LIN {X -0.230,Y -500.560,Z 1588.535,A 0.000,B 0.000,C 90.000,E1 96.372} C_DIS
LIN {X 0.139,Y -499.439,Z 1588.534,A 0.000,B 0.000,C 90.000,E1 96.087} C_DIS
LIN {X -0.151,Y -494.579,Z 1588.530,A 0.000,B 0.000,C 90.000,E1 95.391} C_DIS
LIN {X 0.194,Y -481.570,Z 1588.519,A 0.000,B 0.000,C 90.000,E1 93.383} C_DIS
LIN {X 0.131,Y -471.581,Z 1588.511,A 0.000,B 0.000,C 90.000,E1 91.892} C_DIS
LIN {X 0.103,Y -462.930,Z 1588.504,A 0.000,B 0.000,C 90.000,E1 90.630} C_DIS
LIN {X -0.051,Y -453.933,Z 1588.496,A 0.000,B 0.000,C 90.000,E1 89.370} C_DIS
LIN {X 0.124,Y -444.506,Z 1588.489,A 0.000,B 0.000,C 90.000,E1 88.051} C_DIS
LIN {X -0.111,Y -432.606,Z 1588.480,A 0.000,B 0.000,C 90.000,E1 86.502} C_DIS
LIN {X 0.018,Y -418.492,Z 1588.470,A 0.000,B 0.000,C 90.000,E1 84.609} C_DIS
LIN {X 0.166,Y -399.403,Z 1588.455,A 0.000,B 0.000,C 90.000,E1 81.837} C_DIS
LIN {X -0.155,Y -383.351,Z 1588.441,A 0.000,B 0.000,C 90.000,E1 79.342} C_DIS
LIN {X 0.055,Y -364.882,Z 1588.423,A 0.000,B 0.000,C 90.000,E1 76.117} C_DIS
LIN {X 0.022,Y -351.994,Z 1588.410,A 0.000,B 0.000,C 90.000,E1 73.740} C_DIS
LIN {X -0.111,Y -339.351,Z 1588.396,A 0.000,B 0.000,C 90.000,E1 71.329} C_DIS
LIN {X -0.034,Y -325.790,Z 1588.381,A 0.000,B 0.000,C 90.000,E1 68.518} C_DIS
LIN {X -0.019,Y -314.232,Z 1588.366,A 0.000,B 0.000,C 90.000,E1 65.973} C_DIS
LIN {X -0.119,Y -300.650,Z 1588.348,A 0.000,B 0.000,C 90.000,E1 62.743} C_DIS
LIN {X 0.080,Y -292.540,Z 1588.337,A 0.000,B 0.000,C 90.000,E1 60.717} C_DIS
LIN {X -0.130,Y -284.116,Z 1588.326,A 0.000,B 0.000,C 90.000,E1 58.742} C_DIS
LIN {X 0.132,Y -273.947,Z 1588.313,A 0.000,B 0.000,C 90.000,E1 56.294} C_DIS
LIN {X -0.133,Y -263.749,Z 1588.299,A 0.000,B 0.000,C 90.000,E1 53.909} C_DIS
LIN {X -0.023,Y -251.335,Z 1588.281,A 0.000,B 0.000,C 90.000,E1 50.678} C_DIS
LIN {X -0.018,Y -239.866,Z 1588.263,A 0.000,B 0.000,C 90.000,E1 47.391} C_DIS
LIN {X -0.003,Y -229.485,Z 1588.245,A 0.000,B 0.000,C 90.000,E1 44.028} C_DIS
LIN {X -0.004,Y -221.059,Z 1588.228,A 0.000,B 0.000,C 90.000,E1 40.987} C_DIS
LIN {X 0.009,Y -213.332,Z 1588.211,A 0.000,B 0.000,C 90.000,E1 37.890} C_DIS
LIN {X 0.035,Y -206.409,Z 1588.193,A 0.000,B 0.000,C 90.000,E1 34.739} C_DIS
LIN {X 0.050,Y -200.208,Z 1588.175,A 0.000,B 0.000,C 90.000,E1 31.544} C_DIS
LIN {X 0.055,Y -194.851,Z 1588.157,A 0.000,B 0.000,C 90.000,E1 28.309} C_DIS
LIN {X 0.086,Y -190.223,Z 1588.139,A 0.000,B 0.000,C 90.000,E1 25.027} C_DIS
LIN {X -0.003,Y -185.282,Z 1588.116,A 0.000,B 0.000,C 90.000,E1 20.918} C_DIS
LIN {X 0.013,Y -181.201,Z 1588.093,A 0.000,B 0.000,C 90.000,E1 16.732} C_DIS
LIN {X -0.054,Y -177.876,Z 1588.070,A 0.000,B 0.000,C 90.000,E1 12.535} C_DIS
LIN {X 0.018,Y -175.021,Z 1588.041,A 0.000,B 0.000,C 90.000,E1 7.409} C_DIS
LIN {X -0.025,Y -172.799,Z 1588.008,A 0.000,B 0.000,C 90.000,E1 1.432} C_DIS
LIN {X 0.049,Y -173.988,Z 1587.935,A 0.000,B 0.000,C 90.000,E1 348.342} C_DIS
LIN {X 0.090,Y -176.815,Z 1587.907,A 0.000,B 0.000,C 90.000,E1 343.196} C_DIS
LIN {X 0.073,Y -180.404,Z 1587.883,A 0.000,B 0.000,C 90.000,E1 338.954} C_DIS
LIN {X -0.083,Y -185.209,Z 1587.860,A 0.000,B 0.000,C 90.000,E1 334.793} C_DIS
LIN {X -0.009,Y -189.881,Z 1587.841,A 0.000,B 0.000,C 90.000,E1 331.435} C_DIS
LIN {X 0.040,Y -195.211,Z 1587.823,A 0.000,B 0.000,C 90.000,E1 328.122} C_DIS
LIN {X -0.072,Y -201.335,Z 1587.805,A 0.000,B 0.000,C 90.000,E1 324.895} C_DIS
LIN {X -0.008,Y -208.216,Z 1587.787,A 0.000,B 0.000,C 90.000,E1 321.662} C_DIS
LIN {X 0.040,Y -216.014,Z 1587.769,A 0.000,B 0.000,C 90.000,E1 318.485} C_DIS
LIN {X 0.023,Y -225.787,Z 1587.750,A 0.000,B 0.000,C 90.000,E1 315.000} C_DIS
LIN {X -0.103,Y -234.279,Z 1587.735,A 0.000,B 0.000,C 90.000,E1 312.366} C_DIS
LIN {X 0.012,Y -242.255,Z 1587.723,A 0.000,B 0.000,C 90.000,E1 310.092} C_DIS
LIN {X -0.029,Y -248.230,Z 1587.715,A 0.000,B 0.000,C 90.000,E1 308.624} C_DIS
LIN {X 0.005,Y -254.959,Z 1587.706,A 0.000,B 0.000,C 90.000,E1 307.156} C_DIS
LIN {X 0.013,Y -264.367,Z 1587.696,A 0.000,B 0.000,C 90.000,E1 305.358} C_DIS
LIN {X 0.011,Y -276.846,Z 1587.685,A 0.000,B 0.000,C 90.000,E1 303.245} C_DIS
LIN {X -0.005,Y -293.095,Z 1587.671,A 0.000,B 0.000,C 90.000,E1 300.846} C_DIS
LIN {X 0.122,Y -308.007,Z 1587.660,A 0.000,B 0.000,C 90.000,E1 298.821} C_DIS
LIN {X 0.062,Y -320.406,Z 1587.651,A 0.000,B 0.000,C 90.000,E1 297.206} C_DIS
LIN {X 0.191,Y -332.863,Z 1587.642,A 0.000,B 0.000,C 90.000,E1 295.591} C_DIS
LIN {X -0.075,Y -344.944,Z 1587.634,A 0.000,B 0.000,C 90.000,E1 294.079} C_DIS
LIN {X -0.087,Y -362.411,Z 1587.622,A 0.000,B 0.000,C 90.000,E1 291.950} C_DIS
LIN {X 0.161,Y -374.913,Z 1587.614,A 0.000,B 0.000,C 90.000,E1 290.429} C_DIS
LIN {X 0.128,Y -384.438,Z 1587.607,A 0.000,B 0.000,C 90.000,E1 289.268} C_DIS
LIN {X 0.049,Y -391.088,Z 1587.602,A 0.000,B 0.000,C 90.000,E1 288.417} C_DIS
LIN {X -0.087,Y -397.218,Z 1587.598,A 0.000,B 0.000,C 90.000,E1 287.583} C_DIS
LIN {X 0.148,Y -400.979,Z 1587.594,A 0.000,B 0.000,C 90.000,E1 286.985} C_DIS
LIN {X 0.104,Y -405.869,Z 1587.590,A 0.000,B 0.000,C 90.000,E1 286.150} C_DIS
LIN {X 0.006,Y -408.632,Z 1587.587,A 0.000,B 0.000,C 90.000,E1 285.607} C_DIS
LIN {X -0.077,Y -411.045,Z 1587.584,A 0.000,B 0.000,C 90.000,E1 285.064} C_DIS
LIN {X 0.146,Y -413.036,Z 1587.581,A 0.000,B 0.000,C 90.000,E1 284.481} C_DIS
LIN {X 0.080,Y -414.633,Z 1587.578,A 0.000,B 0.000,C 90.000,E1 283.939} C_DIS
LIN {X -0.077,Y -415.820,Z 1587.574,A 0.000,B 0.000,C 90.000,E1 283.411} C_DIS
LIN {X 0.182,Y -416.599,Z 1587.571,A 0.000,B 0.000,C 90.000,E1 282.827} C_DIS
LIN {X 0.044,Y -416.869,Z 1587.568,A 0.000,B 0.000,C 90.000,E1 282.299} C_DIS
LIN {X -0.090,Y -416.664,Z 1587.565,A 0.000,B 0.000,C 90.000,E1 281.771} C_DIS
LIN {X 0.185,Y -415.926,Z 1587.562,A 0.000,B 0.000,C 90.000,E1 281.186} C_DIS
LIN {X 0.049,Y -414.668,Z 1587.559,A 0.000,B 0.000,C 90.000,E1 280.658} C_DIS
LIN {X -0.165,Y -412.786,Z 1587.556,A 0.000,B 0.000,C 90.000,E1 280.141} C_DIS
LIN {X 0.094,Y -410.280,Z 1587.553,A 0.000,B 0.000,C 90.000,E1 279.557} C_DIS
LIN {X -0.073,Y -407.020,Z 1587.550,A 0.000,B 0.000,C 90.000,E1 279.029} C_DIS
LIN {X -0.026,Y -405.197,Z 1587.549,A 0.000,B 0.000,C 90.000,E1 278.746} C_DIS
LIN {X 0.177,Y -400.827,Z 1587.546,A 0.000,B 0.000,C 90.000,E1 278.163} C_DIS
LIN {X -0.097,Y -395.813,Z 1587.542,A 0.000,B 0.000,C 90.000,E1 277.644} C_DIS
LIN {X 0.138,Y -390.224,Z 1587.539,A 0.000,B 0.000,C 90.000,E1 277.068} C_DIS
LIN {X -0.161,Y -384.400,Z 1587.537,A 0.000,B 0.000,C 90.000,E1 276.606} C_DIS
LIN {X 0.160,Y -378.276,Z 1587.534,A 0.000,B 0.000,C 90.000,E1 276.087} C_DIS
LIN {X 0.005,Y -371.989,Z 1587.532,A 0.000,B 0.000,C 90.000,E1 275.682} C_DIS
LIN {X 0.032,Y -362.421,Z 1587.528,A 0.000,B 0.000,C 90.000,E1 275.106} C_DIS
LIN {X 0.140,Y -352.870,Z 1587.526,A 0.000,B 0.000,C 90.000,E1 274.588} C_DIS
LIN {X 0.138,Y -343.087,Z 1587.523,A 0.000,B 0.000,C 90.000,E1 274.131} C_DIS
LIN {X 0.113,Y -333.414,Z 1587.521,A 0.000,B 0.000,C 90.000,E1 273.726} C_DIS
LIN {X -0.095,Y -320.424,Z 1587.518,A 0.000,B 0.000,C 90.000,E1 273.269} C_DIS
LIN {X -0.022,Y -310.456,Z 1587.516,A 0.000,B 0.000,C 90.000,E1 272.922} C_DIS
LIN {X -0.024,Y -299.914,Z 1587.515,A 0.000,B 0.000,C 90.000,E1 272.636} C_DIS
LIN {X 0.033,Y -292.289,Z 1587.514,A 0.000,B 0.000,C 90.000,E1 272.465} C_DIS
LIN {X -0.085,Y -279.300,Z 1587.513,A 0.000,B 0.000,C 90.000,E1 272.293} C_DIS
LIN {X -0.016,Y -260.975,Z 1587.511,A 0.000,B 0.000,C 90.000,E1 272.064} C_DIS
LIN {X -0.040,Y -244.011,Z 1587.511,A 0.000,B 0.000,C 90.000,E1 271.949} C_DIS
LIN {X 0.107,Y -235.308,Z 1587.511,A 0.000,B 0.000,C 90.000,E1 271.892} C_DIS
LIN {X 0.048,Y -181.277,Z 1587.511,A 0.000,B 0.000,C 90.000,E1 271.892} C_DIS
LIN {X 0.057,Y -181.579,Z 1587.501,A 0.000,B 0.000,C 90.000,E1 270.172} C_DIS
LIN {X 0.045,Y -180.887,Z 1587.473,A 0.000,B 0.000,C 90.000,E1 265.122} C_DIS
LIN {X -0.072,Y -179.010,Z 1587.445,A 0.000,B 0.000,C 90.000,E1 260.095} C_DIS
LIN {X 0.023,Y -178.625,Z 1587.440,A 0.000,B 0.000,C 90.000,E1 259.218} C_DIS
LIN {X -0.079,Y -175.676,Z 1587.412,A 0.000,B 0.000,C 90.000,E1 254.157} C_DIS
LIN {X -0.067,Y -172.393,Z 1587.388,A 0.000,B 0.000,C 90.000,E1 249.880} C_DIS
LIN {X -0.050,Y -171.199,Z 1587.379,A 0.000,B 0.000,C 90.000,E1 248.156} C_DIS
LIN {X 0.001,Y -167.488,Z 1587.355,A 0.000,B 0.000,C 90.000,E1 243.819} C_DIS
LIN {X 0.009,Y -166.884,Z 1587.350,A 0.000,B 0.000,C 90.000,E1 242.948} C_DIS
LIN {X 0.000,Y -162.189,Z 1587.321,A 0.000,B 0.000,C 90.000,E1 237.709} C_DIS
LIN {X -0.033,Y -160.758,Z 1587.311,A 0.000,B 0.000,C 90.000,E1 235.960} C_DIS
LIN {X 0.036,Y -157.555,Z 1587.291,A 0.000,B 0.000,C 90.000,E1 232.396} C_DIS
LIN {X -0.027,Y -155.584,Z 1587.276,A 0.000,B 0.000,C 90.000,E1 229.747} C_DIS
LIN {X 0.025,Y -151.869,Z 1587.251,A 0.000,B 0.000,C 90.000,E1 225.243} C_DIS
LIN {X 0.039,Y -150.093,Z 1587.236,A 0.000,B 0.000,C 90.000,E1 222.528} C_DIS
LIN {X -0.044,Y -146.893,Z 1587.211,A 0.000,B 0.000,C 90.000,E1 218.016} C_DIS
LIN {X 0.061,Y -145.480,Z 1587.196,A 0.000,B 0.000,C 90.000,E1 215.231} C_DIS
LIN {X -0.023,Y -142.889,Z 1587.170,A 0.000,B 0.000,C 90.000,E1 210.669} C_DIS
LIN {X 0.034,Y -141.509,Z 1587.150,A 0.000,B 0.000,C 90.000,E1 206.950} C_DIS
LIN {X -0.049,Y -139.391,Z 1587.114,A 0.000,B 0.000,C 90.000,E1 200.482} C_DIS
LIN {X 0.003,Y -139.100,Z 1587.103,A 0.000,B 0.000,C 90.000,E1 198.598} C_DIS
LIN {X -0.006,Y -138.353,Z 1587.057,A 0.000,B 0.000,C 90.000,E1 190.197} C_DIS
LIN {X -0.012,Y -139.515,Z 1587.005,A 0.000,B 0.000,C 90.000,E1 180.859} C_DIS
LIN {X -0.072,Y -141.166,Z 1586.974,A 0.000,B 0.000,C 90.000,E1 175.298} C_DIS
LIN {X 0.040,Y -142.545,Z 1586.958,A 0.000,B 0.000,C 90.000,E1 172.470} C_DIS
LIN {X -0.035,Y -144.819,Z 1586.933,A 0.000,B 0.000,C 90.000,E1 167.881} C_DIS
LIN {X -0.048,Y -147.440,Z 1586.912,A 0.000,B 0.000,C 90.000,E1 164.212} C_DIS
LIN {X -0.019,Y -150.020,Z 1586.892,A 0.000,B 0.000,C 90.000,E1 160.550} C_DIS
LIN {X -0.013,Y -153.355,Z 1586.872,A 0.000,B 0.000,C 90.000,E1 156.922} C_DIS
LIN {X 0.036,Y -155.889,Z 1586.857,A 0.000,B 0.000,C 90.000,E1 154.204} C_DIS
LIN {X -0.066,Y -159.746,Z 1586.837,A 0.000,B 0.000,C 90.000,E1 150.667} C_DIS
LIN {X 0.000,Y -161.987,Z 1586.827,A 0.000,B 0.000,C 90.000,E1 148.869} C_DIS
LIN {X 0.020,Y -166.179,Z 1586.807,A 0.000,B 0.000,C 90.000,E1 145.341} C_DIS
LIN {X 0.013,Y -171.193,Z 1586.788,A 0.000,B 0.000,C 90.000,E1 141.859} C_DIS
LIN {X 0.043,Y -176.076,Z 1586.769,A 0.000,B 0.000,C 90.000,E1 138.405} C_DIS
LIN {X -0.094,Y -180.335,Z 1586.755,A 0.000,B 0.000,C 90.000,E1 135.891} C_DIS
LIN {X 0.014,Y -185.744,Z 1586.736,A 0.000,B 0.000,C 90.000,E1 132.486} C_DIS
LIN {X -0.073,Y -190.355,Z 1586.722,A 0.000,B 0.000,C 90.000,E1 130.011} C_DIS
LIN {X -0.026,Y -197.681,Z 1586.699,A 0.000,B 0.000,C 90.000,E1 125.884} C_DIS
LIN {X 0.015,Y -200.933,Z 1586.690,A 0.000,B 0.000,C 90.000,E1 124.246} C_DIS
LIN {X 0.074,Y -204.518,Z 1586.679,A 0.000,B 0.000,C 90.000,E1 122.212} C_DIS
LIN {X 0.056,Y -322.284,Z 1586.679,A 0.000,B 0.000,C 90.000,E1 122.212} C_DIS
LIN {X -0.123,Y -323.983,Z 1586.679,A 0.000,B 0.000,C 90.000,E1 122.212} C_DIS
LIN {X 0.034,Y -327.982,Z 1586.678,A 0.000,B 0.000,C 90.000,E1 122.005} C_DIS
LIN {X 0.193,Y -330.311,Z 1586.677,A 0.000,B 0.000,C 90.000,E1 121.799} C_DIS
LIN {X -0.018,Y -334.169,Z 1586.674,A 0.000,B 0.000,C 90.000,E1 121.386} C_DIS
LIN {X 0.129,Y -336.011,Z 1586.673,A 0.000,B 0.000,C 90.000,E1 121.052} C_DIS
LIN {X -0.047,Y -338.678,Z 1586.669,A 0.000,B 0.000,C 90.000,E1 120.463} C_DIS
LIN {X -0.038,Y -350.483,Z 1586.654,A 0.000,B 0.000,C 90.000,E1 117.692} C_DIS
LIN {X 0.139,Y -363.724,Z 1586.639,A 0.000,B 0.000,C 90.000,E1 114.951} C_DIS
LIN {X -0.094,Y -378.522,Z 1586.624,A 0.000,B 0.000,C 90.000,E1 112.333} C_DIS
LIN {X 0.143,Y -393.083,Z 1586.611,A 0.000,B 0.000,C 90.000,E1 109.993} C_DIS
LIN {X -0.023,Y -409.073,Z 1586.599,A 0.000,B 0.000,C 90.000,E1 107.764} C_DIS
LIN {X 0.089,Y -426.603,Z 1586.586,A 0.000,B 0.000,C 90.000,E1 105.552} C_DIS
LIN {X 0.128,Y -445.761,Z 1586.575,A 0.000,B 0.000,C 90.000,E1 103.411} C_DIS
LIN {X 0.086,Y -465.835,Z 1586.563,A 0.000,B 0.000,C 90.000,E1 101.422} C_DIS
LIN {X 0.034,Y -489.042,Z 1586.552,A 0.000,B 0.000,C 90.000,E1 99.378} C_DIS
LIN {X -0.187,Y -494.277,Z 1586.550,A 0.000,B 0.000,C 90.000,E1 98.973} C_DIS
LIN {X -0.072,Y -496.442,Z 1586.549,A 0.000,B 0.000,C 90.000,E1 98.746} C_DIS
LIN {X -0.113,Y -498.267,Z 1586.547,A 0.000,B 0.000,C 90.000,E1 98.511} C_DIS
LIN {X -0.155,Y -499.640,Z 1586.546,A 0.000,B 0.000,C 90.000,E1 98.276} C_DIS
LIN {X 0.118,Y -501.397,Z 1586.543,A 0.000,B 0.000,C 90.000,E1 97.757} C_DIS
LIN {X -0.098,Y -502.041,Z 1586.541,A 0.000,B 0.000,C 90.000,E1 97.296} C_DIS
LIN {X 0.195,Y -501.682,Z 1586.538,A 0.000,B 0.000,C 90.000,E1 96.777} C_DIS
LIN {X -0.006,Y -500.267,Z 1586.535,A 0.000,B 0.000,C 90.000,E1 96.315} C_DIS
LIN {X -0.133,Y -499.089,Z 1586.534,A 0.000,B 0.000,C 90.000,E1 96.087} C_DIS
LIN {X -0.126,Y -486.046,Z 1586.523,A 0.000,B 0.000,C 90.000,E1 94.131} C_DIS
LIN {X -0.083,Y -476.250,Z 1586.515,A 0.000,B 0.000,C 90.000,E1 92.636} C_DIS
LIN {X 0.231,Y -466.095,Z 1586.506,A 0.000,B 0.000,C 90.000,E1 91.088} C_DIS
LIN {X -0.105,Y -455.371,Z 1586.498,A 0.000,B 0.000,C 90.000,E1 89.599} C_DIS
LIN {X 0.083,Y -446.043,Z 1586.490,A 0.000,B 0.000,C 90.000,E1 88.282} C_DIS
LIN {X 0.135,Y -436.232,Z 1586.483,A 0.000,B 0.000,C 90.000,E1 86.963} C_DIS
LIN {X -0.059,Y -422.140,Z 1586.473,A 0.000,B 0.000,C 90.000,E1 85.122} C_DIS
LIN {X -0.198,Y -400.891,Z 1586.456,A 0.000,B 0.000,C 90.000,E1 82.129} C_DIS
LIN {X -0.047,Y -383.024,Z 1586.440,A 0.000,B 0.000,C 90.000,E1 79.285} C_DIS
LIN {X 0.144,Y -364.572,Z 1586.423,A 0.000,B 0.000,C 90.000,E1 76.061} C_DIS
LIN {X 0.095,Y -351.683,Z 1586.409,A 0.000,B 0.000,C 90.000,E1 73.685} C_DIS
LIN {X -0.051,Y -339.047,Z 1586.396,A 0.000,B 0.000,C 90.000,E1 71.275} C_DIS
LIN {X 0.009,Y -325.528,Z 1586.380,A 0.000,B 0.000,C 90.000,E1 68.465} C_DIS
LIN {X 0.011,Y -313.943,Z 1586.366,A 0.000,B 0.000,C 90.000,E1 65.921} C_DIS
LIN {X 0.009,Y -301.647,Z 1586.350,A 0.000,B 0.000,C 90.000,E1 62.999} C_DIS
LIN {X 0.081,Y -293.519,Z 1586.339,A 0.000,B 0.000,C 90.000,E1 61.001} C_DIS
LIN {X 0.030,Y -285.091,Z 1586.328,A 0.000,B 0.000,C 90.000,E1 58.997} C_DIS
LIN {X -0.021,Y -276.443,Z 1586.316,A 0.000,B 0.000,C 90.000,E1 56.962} C_DIS
LIN {X -0.004,Y -266.311,Z 1586.303,A 0.000,B 0.000,C 90.000,E1 54.529} C_DIS
LIN {X 0.022,Y -253.756,Z 1586.285,A 0.000,B 0.000,C 90.000,E1 51.331} C_DIS
LIN {X -0.066,Y -242.103,Z 1586.267,A 0.000,B 0.000,C 90.000,E1 48.081} C_DIS
LIN {X 0.015,Y -231.529,Z 1586.248,A 0.000,B 0.000,C 90.000,E1 44.717} C_DIS
LIN {X 0.052,Y -222.941,Z 1586.232,A 0.000,B 0.000,C 90.000,E1 41.676} C_DIS
LIN {X -0.057,Y -215.065,Z 1586.214,A 0.000,B 0.000,C 90.000,E1 38.624} C_DIS
LIN {X 0.019,Y -207.965,Z 1586.197,A 0.000,B 0.000,C 90.000,E1 35.471} C_DIS
LIN {X 0.020,Y -201.641,Z 1586.179,A 0.000,B 0.000,C 90.000,E1 32.291} C_DIS
LIN {X -0.013,Y -196.095,Z 1586.161,A 0.000,B 0.000,C 90.000,E1 29.077} C_DIS
LIN {X 0.049,Y -191.343,Z 1586.143,A 0.000,B 0.000,C 90.000,E1 25.796} C_DIS
LIN {X -0.102,Y -186.255,Z 1586.120,A 0.000,B 0.000,C 90.000,E1 21.716} C_DIS
LIN {X 0.006,Y -182.052,Z 1586.097,A 0.000,B 0.000,C 90.000,E1 17.511} C_DIS
LIN {X 0.009,Y -178.605,Z 1586.074,A 0.000,B 0.000,C 90.000,E1 13.300} C_DIS
LIN {X -0.034,Y -175.596,Z 1586.046,A 0.000,B 0.000,C 90.000,E1 8.219} C_DIS
LIN {X -0.039,Y -173.470,Z 1586.017,A 0.000,B 0.000,C 90.000,E1 3.094} C_DIS
LIN {X 0.066,Y -174.236,Z 1585.935,A 0.000,B 0.000,C 90.000,E1 348.342} C_DIS
LIN {X -0.052,Y -177.058,Z 1585.907,A 0.000,B 0.000,C 90.000,E1 343.251} C_DIS
LIN {X 0.045,Y -180.646,Z 1585.883,A 0.000,B 0.000,C 90.000,E1 338.975} C_DIS
LIN {X -0.040,Y -185.422,Z 1585.860,A 0.000,B 0.000,C 90.000,E1 334.793} C_DIS
LIN {X 0.041,Y -190.093,Z 1585.841,A 0.000,B 0.000,C 90.000,E1 331.435} C_DIS
LIN {X 0.097,Y -195.382,Z 1585.823,A 0.000,B 0.000,C 90.000,E1 328.122} C_DIS
LIN {X -0.009,Y -201.459,Z 1585.805,A 0.000,B 0.000,C 90.000,E1 324.895} C_DIS
LIN {X -0.069,Y -208.332,Z 1585.787,A 0.000,B 0.000,C 90.000,E1 321.698} C_DIS
LIN {X -0.055,Y -216.110,Z 1585.770,A 0.000,B 0.000,C 90.000,E1 318.528} C_DIS
LIN {X 0.013,Y -224.671,Z 1585.752,A 0.000,B 0.000,C 90.000,E1 315.405} C_DIS
LIN {X -0.135,Y -232.992,Z 1585.737,A 0.000,B 0.000,C 90.000,E1 312.771} C_DIS
LIN {X 0.090,Y -242.189,Z 1585.723,A 0.000,B 0.000,C 90.000,E1 310.092} C_DIS
LIN {X 0.050,Y -248.139,Z 1585.715,A 0.000,B 0.000,C 90.000,E1 308.624} C_DIS
LIN {X 0.084,Y -254.849,Z 1585.707,A 0.000,B 0.000,C 90.000,E1 307.156} C_DIS
LIN {X -0.059,Y -264.221,Z 1585.697,A 0.000,B 0.000,C 90.000,E1 305.391} C_DIS
LIN {X -0.138,Y -276.694,Z 1585.685,A 0.000,B 0.000,C 90.000,E1 303.293} C_DIS
LIN {X -0.045,Y -290.496,Z 1585.673,A 0.000,B 0.000,C 90.000,E1 301.209} C_DIS
LIN {X -0.080,Y -305.332,Z 1585.662,A 0.000,B 0.000,C 90.000,E1 299.205} C_DIS
LIN {X -0.053,Y -317.780,Z 1585.653,A 0.000,B 0.000,C 90.000,E1 297.564} C_DIS
LIN {X -0.023,Y -332.733,Z 1585.642,A 0.000,B 0.000,C 90.000,E1 295.643} C_DIS
LIN {X 0.014,Y -342.443,Z 1585.635,A 0.000,B 0.000,C 90.000,E1 294.387} C_DIS
LIN {X 0.002,Y -362.352,Z 1585.622,A 0.000,B 0.000,C 90.000,E1 291.950} C_DIS
LIN {X -0.099,Y -374.901,Z 1585.614,A 0.000,B 0.000,C 90.000,E1 290.482} C_DIS
LIN {X 0.092,Y -382.181,Z 1585.609,A 0.000,B 0.000,C 90.000,E1 289.577} C_DIS
LIN {X 0.002,Y -389.025,Z 1585.604,A 0.000,B 0.000,C 90.000,E1 288.725} C_DIS
LIN {X -0.038,Y -395.368,Z 1585.599,A 0.000,B 0.000,C 90.000,E1 287.873} C_DIS
LIN {X -0.136,Y -401.153,Z 1585.595,A 0.000,B 0.000,C 90.000,E1 287.040} C_DIS
LIN {X -0.184,Y -406.094,Z 1585.590,A 0.000,B 0.000,C 90.000,E1 286.205} C_DIS
LIN {X -0.181,Y -410.131,Z 1585.585,A 0.000,B 0.000,C 90.000,E1 285.371} C_DIS
LIN {X -0.146,Y -413.313,Z 1585.581,A 0.000,B 0.000,C 90.000,E1 284.537} C_DIS
LIN {X 0.096,Y -414.931,Z 1585.578,A 0.000,B 0.000,C 90.000,E1 283.953} C_DIS
LIN {X 0.041,Y -416.180,Z 1585.575,A 0.000,B 0.000,C 90.000,E1 283.411} C_DIS
LIN {X -0.104,Y -416.959,Z 1585.572,A 0.000,B 0.000,C 90.000,E1 282.883} C_DIS
LIN {X 0.166,Y -417.295,Z 1585.568,A 0.000,B 0.000,C 90.000,E1 282.299} C_DIS
LIN {X 0.034,Y -417.100,Z 1585.565,A 0.000,B 0.000,C 90.000,E1 281.771} C_DIS
LIN {X -0.096,Y -416.420,Z 1585.562,A 0.000,B 0.000,C 90.000,E1 281.243} C_DIS
LIN {X 0.178,Y -415.171,Z 1585.559,A 0.000,B 0.000,C 90.000,E1 280.658} C_DIS
LIN {X -0.034,Y -413.359,Z 1585.556,A 0.000,B 0.000,C 90.000,E1 280.141} C_DIS
LIN {X -0.177,Y -410.846,Z 1585.553,A 0.000,B 0.000,C 90.000,E1 279.613} C_DIS
LIN {X 0.063,Y -407.644,Z 1585.550,A 0.000,B 0.000,C 90.000,E1 279.029} C_DIS
LIN {X -0.181,Y -403.766,Z 1585.547,A 0.000,B 0.000,C 90.000,E1 278.511} C_DIS
LIN {X -0.041,Y -399.179,Z 1585.544,A 0.000,B 0.000,C 90.000,E1 277.936} C_DIS
LIN {X 0.125,Y -393.746,Z 1585.541,A 0.000,B 0.000,C 90.000,E1 277.352} C_DIS
LIN {X 0.044,Y -387.981,Z 1585.538,A 0.000,B 0.000,C 90.000,E1 276.834} C_DIS
LIN {X -0.109,Y -382.050,Z 1585.535,A 0.000,B 0.000,C 90.000,E1 276.372} C_DIS
LIN {X -0.044,Y -375.775,Z 1585.533,A 0.000,B 0.000,C 90.000,E1 275.910} C_DIS
LIN {X -0.133,Y -366.366,Z 1585.530,A 0.000,B 0.000,C 90.000,E1 275.334} C_DIS
LIN {X 0.143,Y -360.036,Z 1585.528,A 0.000,B 0.000,C 90.000,E1 274.935} C_DIS
LIN {X -0.012,Y -350.334,Z 1585.525,A 0.000,B 0.000,C 90.000,E1 274.473} C_DIS
LIN {X 0.133,Y -340.680,Z 1585.522,A 0.000,B 0.000,C 90.000,E1 274.012} C_DIS
LIN {X 0.130,Y -324.911,Z 1585.519,A 0.000,B 0.000,C 90.000,E1 273.383} C_DIS
LIN {X 0.094,Y -314.863,Z 1585.517,A 0.000,B 0.000,C 90.000,E1 273.037} C_DIS
LIN {X -0.054,Y -304.256,Z 1585.515,A 0.000,B 0.000,C 90.000,E1 272.751} C_DIS
LIN {X 0.141,Y -293.526,Z 1585.514,A 0.000,B 0.000,C 90.000,E1 272.465} C_DIS
LIN {X 0.012,Y -280.763,Z 1585.513,A 0.000,B 0.000,C 90.000,E1 272.293} C_DIS
LIN {X 0.057,Y -262.332,Z 1585.511,A 0.000,B 0.000,C 90.000,E1 272.064} C_DIS
LIN {X 0.031,Y -246.556,Z 1585.511,A 0.000,B 0.000,C 90.000,E1 271.949} C_DIS
LIN {X -0.102,Y -232.708,Z 1585.511,A 0.000,B 0.000,C 90.000,E1 271.949} C_DIS
LIN {X 0.067,Y -181.276,Z 1585.511,A 0.000,B 0.000,C 90.000,E1 271.892} C_DIS
LIN {X -0.070,Y -181.580,Z 1585.501,A 0.000,B 0.000,C 90.000,E1 270.229} C_DIS
LIN {X -0.080,Y -180.890,Z 1585.473,A 0.000,B 0.000,C 90.000,E1 265.179} C_DIS
LIN {X -0.018,Y -179.013,Z 1585.445,A 0.000,B 0.000,C 90.000,E1 260.095} C_DIS
LIN {X 0.076,Y -178.637,Z 1585.440,A 0.000,B 0.000,C 90.000,E1 259.218} C_DIS
LIN {X -0.026,Y -175.688,Z 1585.412,A 0.000,B 0.000,C 90.000,E1 254.157} C_DIS
LIN {X -0.015,Y -172.404,Z 1585.388,A 0.000,B 0.000,C 90.000,E1 249.880} C_DIS
LIN {X 0.002,Y -171.216,Z 1585.379,A 0.000,B 0.000,C 90.000,E1 248.156} C_DIS
LIN {X -0.021,Y -167.500,Z 1585.355,A 0.000,B 0.000,C 90.000,E1 243.845} C_DIS
LIN {X -0.089,Y -166.896,Z 1585.350,A 0.000,B 0.000,C 90.000,E1 242.999} C_DIS
LIN {X -0.036,Y -162.202,Z 1585.321,A 0.000,B 0.000,C 90.000,E1 237.740} C_DIS
LIN {X 0.017,Y -160.777,Z 1585.311,A 0.000,B 0.000,C 90.000,E1 235.960} C_DIS
LIN {X -0.011,Y -157.570,Z 1585.291,A 0.000,B 0.000,C 90.000,E1 232.431} C_DIS
LIN {X 0.023,Y -155.601,Z 1585.276,A 0.000,B 0.000,C 90.000,E1 229.747} C_DIS
LIN {X 0.073,Y -151.882,Z 1585.251,A 0.000,B 0.000,C 90.000,E1 225.243} C_DIS
LIN {X 0.087,Y -150.108,Z 1585.236,A 0.000,B 0.000,C 90.000,E1 222.528} C_DIS
LIN {X 0.004,Y -146.904,Z 1585.211,A 0.000,B 0.000,C 90.000,E1 218.016} C_DIS
LIN {X 0.024,Y -145.491,Z 1585.196,A 0.000,B 0.000,C 90.000,E1 215.264} C_DIS
LIN {X 0.024,Y -142.897,Z 1585.170,A 0.000,B 0.000,C 90.000,E1 210.669} C_DIS
LIN {X -0.045,Y -141.518,Z 1585.150,A 0.000,B 0.000,C 90.000,E1 207.001} C_DIS
LIN {X -0.002,Y -139.395,Z 1585.114,A 0.000,B 0.000,C 90.000,E1 200.482} C_DIS
LIN {X 0.048,Y -139.105,Z 1585.103,A 0.000,B 0.000,C 90.000,E1 198.598} C_DIS
LIN {X 0.040,Y -138.353,Z 1585.057,A 0.000,B 0.000,C 90.000,E1 190.197} C_DIS
LIN {X 0.034,Y -139.511,Z 1585.005,A 0.000,B 0.000,C 90.000,E1 180.859} C_DIS
LIN {X -0.025,Y -141.157,Z 1584.974,A 0.000,B 0.000,C 90.000,E1 175.298} C_DIS
LIN {X -0.055,Y -142.537,Z 1584.958,A 0.000,B 0.000,C 90.000,E1 172.527} C_DIS
LIN {X 0.013,Y -144.807,Z 1584.933,A 0.000,B 0.000,C 90.000,E1 167.881} C_DIS
LIN {X 0.001,Y -147.427,Z 1584.912,A 0.000,B 0.000,C 90.000,E1 164.212} C_DIS
LIN {X 0.029,Y -150.005,Z 1584.892,A 0.000,B 0.000,C 90.000,E1 160.550} C_DIS
LIN {X 0.037,Y -153.336,Z 1584.872,A 0.000,B 0.000,C 90.000,E1 156.922} C_DIS
LIN {X 0.018,Y -155.871,Z 1584.857,A 0.000,B 0.000,C 90.000,E1 154.229} C_DIS
LIN {X -0.016,Y -159.725,Z 1584.837,A 0.000,B 0.000,C 90.000,E1 150.667} C_DIS
LIN {X 0.052,Y -161.964,Z 1584.827,A 0.000,B 0.000,C 90.000,E1 148.869} C_DIS
LIN {X -0.065,Y -166.155,Z 1584.808,A 0.000,B 0.000,C 90.000,E1 145.388} C_DIS
LIN {X -0.069,Y -171.168,Z 1584.788,A 0.000,B 0.000,C 90.000,E1 141.904} C_DIS
LIN {X -0.035,Y -176.048,Z 1584.769,A 0.000,B 0.000,C 90.000,E1 138.447} C_DIS
LIN {X -0.040,Y -180.304,Z 1584.755,A 0.000,B 0.000,C 90.000,E1 135.891} C_DIS
LIN {X -0.068,Y -185.715,Z 1584.736,A 0.000,B 0.000,C 90.000,E1 132.528} C_DIS
LIN {X -0.017,Y -190.323,Z 1584.722,A 0.000,B 0.000,C 90.000,E1 130.011} C_DIS
LIN {X 0.031,Y -197.649,Z 1584.699,A 0.000,B 0.000,C 90.000,E1 125.884} C_DIS
LIN {X -0.040,Y -200.904,Z 1584.690,A 0.000,B 0.000,C 90.000,E1 124.278} C_DIS
LIN {X 0.022,Y -204.454,Z 1584.679,A 0.000,B 0.000,C 90.000,E1 122.260} C_DIS
LIN {X 0.002,Y -321.406,Z 1584.679,A 0.000,B 0.000,C 90.000,E1 122.260} C_DIS
LIN {X -0.064,Y -322.574,Z 1584.679,A 0.000,B 0.000,C 90.000,E1 122.260} C_DIS
LIN {X -0.029,Y -327.754,Z 1584.678,A 0.000,B 0.000,C 90.000,E1 122.054} C_DIS
LIN {X -0.167,Y -330.353,Z 1584.677,A 0.000,B 0.000,C 90.000,E1 121.878} C_DIS
LIN {X 0.072,Y -334.151,Z 1584.674,A 0.000,B 0.000,C 90.000,E1 121.386} C_DIS
LIN {X 0.024,Y -335.979,Z 1584.673,A 0.000,B 0.000,C 90.000,E1 121.082} C_DIS
LIN {X -0.002,Y -338.626,Z 1584.669,A 0.000,B 0.000,C 90.000,E1 120.463} C_DIS
LIN {X -0.155,Y -350.426,Z 1584.654,A 0.000,B 0.000,C 90.000,E1 117.719} C_DIS
LIN {X 0.031,Y -363.662,Z 1584.639,A 0.000,B 0.000,C 90.000,E1 114.975} C_DIS
LIN {X -0.048,Y -378.456,Z 1584.624,A 0.000,B 0.000,C 90.000,E1 112.333} C_DIS
LIN {X 0.189,Y -393.013,Z 1584.611,A 0.000,B 0.000,C 90.000,E1 109.993} C_DIS
LIN {X 0.024,Y -408.998,Z 1584.599,A 0.000,B 0.000,C 90.000,E1 107.764} C_DIS
LIN {X 0.137,Y -426.523,Z 1584.587,A 0.000,B 0.000,C 90.000,E1 105.552} C_DIS
LIN {X 0.174,Y -445.677,Z 1584.575,A 0.000,B 0.000,C 90.000,E1 103.411} C_DIS
LIN {X 0.129,Y -465.749,Z 1584.564,A 0.000,B 0.000,C 90.000,E1 101.422} C_DIS
LIN {X 0.075,Y -488.955,Z 1584.552,A 0.000,B 0.000,C 90.000,E1 99.378} C_DIS
LIN {X -0.148,Y -494.187,Z 1584.550,A 0.000,B 0.000,C 90.000,E1 98.973} C_DIS
LIN {X -0.033,Y -496.343,Z 1584.549,A 0.000,B 0.000,C 90.000,E1 98.746} C_DIS
LIN {X -0.078,Y -498.165,Z 1584.547,A 0.000,B 0.000,C 90.000,E1 98.511} C_DIS
LIN {X -0.126,Y -499.535,Z 1584.546,A 0.000,B 0.000,C 90.000,E1 98.276} C_DIS
LIN {X 0.146,Y -501.281,Z 1584.543,A 0.000,B 0.000,C 90.000,E1 97.757} C_DIS
LIN {X -0.071,Y -501.915,Z 1584.541,A 0.000,B 0.000,C 90.000,E1 97.296} C_DIS
LIN {X 0.222,Y -501.548,Z 1584.538,A 0.000,B 0.000,C 90.000,E1 96.777} C_DIS
LIN {X 0.020,Y -500.123,Z 1584.535,A 0.000,B 0.000,C 90.000,E1 96.315} C_DIS
LIN {X -0.108,Y -498.939,Z 1584.534,A 0.000,B 0.000,C 90.000,E1 96.087} C_DIS
LIN {X 0.099,Y -482.680,Z 1584.520,A 0.000,B 0.000,C 90.000,E1 93.612} C_DIS
LIN {X 0.054,Y -472.765,Z 1584.512,A 0.000,B 0.000,C 90.000,E1 92.121} C_DIS
LIN {X 0.049,Y -464.198,Z 1584.505,A 0.000,B 0.000,C 90.000,E1 90.859} C_DIS
LIN {X -0.091,Y -455.249,Z 1584.498,A 0.000,B 0.000,C 90.000,E1 89.599} C_DIS
LIN {X 0.095,Y -445.919,Z 1584.490,A 0.000,B 0.000,C 90.000,E1 88.282} C_DIS
LIN {X 0.145,Y -436.137,Z 1584.483,A 0.000,B 0.000,C 90.000,E1 86.963} C_DIS
LIN {X -0.051,Y -422.055,Z 1584.473,A 0.000,B 0.000,C 90.000,E1 85.122} C_DIS
LIN {X -0.100,Y -398.987,Z 1584.455,A 0.000,B 0.000,C 90.000,E1 81.837} C_DIS
LIN {X -0.005,Y -381.225,Z 1584.439,A 0.000,B 0.000,C 90.000,E1 78.993} C_DIS
LIN {X 0.143,Y -364.492,Z 1584.423,A 0.000,B 0.000,C 90.000,E1 76.061} C_DIS
LIN {X 0.150,Y -353.187,Z 1584.411,A 0.000,B 0.000,C 90.000,E1 73.976} C_DIS
LIN {X -0.064,Y -340.523,Z 1584.398,A 0.000,B 0.000,C 90.000,E1 71.583} C_DIS
LIN {X 0.039,Y -326.935,Z 1584.382,A 0.000,B 0.000,C 90.000,E1 68.773} C_DIS
LIN {X 0.073,Y -315.300,Z 1584.368,A 0.000,B 0.000,C 90.000,E1 66.230} C_DIS
LIN {X -0.001,Y -301.497,Z 1584.350,A 0.000,B 0.000,C 90.000,E1 62.999} C_DIS
LIN {X 0.069,Y -293.321,Z 1584.339,A 0.000,B 0.000,C 90.000,E1 61.001} C_DIS
LIN {X 0.014,Y -284.886,Z 1584.328,A 0.000,B 0.000,C 90.000,E1 58.997} C_DIS
LIN {X -0.040,Y -276.256,Z 1584.316,A 0.000,B 0.000,C 90.000,E1 56.962} C_DIS
LIN {X -0.101,Y -267.621,Z 1584.305,A 0.000,B 0.000,C 90.000,E1 54.895} C_DIS
LIN {X -0.040,Y -255.036,Z 1584.287,A 0.000,B 0.000,C 90.000,E1 51.698} C_DIS
LIN {X 0.097,Y -243.345,Z 1584.269,A 0.000,B 0.000,C 90.000,E1 48.405} C_DIS
LIN {X 0.034,Y -232.639,Z 1584.250,A 0.000,B 0.000,C 90.000,E1 45.081} C_DIS
LIN {X 0.029,Y -222.937,Z 1584.232,A 0.000,B 0.000,C 90.000,E1 41.676} C_DIS
LIN {X -0.079,Y -215.084,Z 1584.214,A 0.000,B 0.000,C 90.000,E1 38.624} C_DIS
LIN {X -0.002,Y -207.998,Z 1584.197,A 0.000,B 0.000,C 90.000,E1 35.471} C_DIS
LIN {X 0.000,Y -201.698,Z 1584.179,A 0.000,B 0.000,C 90.000,E1 32.291} C_DIS
LIN {X -0.030,Y -196.181,Z 1584.161,A 0.000,B 0.000,C 90.000,E1 29.077} C_DIS
LIN {X 0.033,Y -190.373,Z 1584.139,A 0.000,B 0.000,C 90.000,E1 24.975} C_DIS
LIN {X 0.022,Y -185.478,Z 1584.116,A 0.000,B 0.000,C 90.000,E1 20.844} C_DIS
LIN {X -0.017,Y -181.461,Z 1584.093,A 0.000,B 0.000,C 90.000,E1 16.677} C_DIS
LIN {X 0.057,Y -177.640,Z 1584.064,A 0.000,B 0.000,C 90.000,E1 11.591} C_DIS
LIN {X 0.058,Y -175.000,Z 1584.036,A 0.000,B 0.000,C 90.000,E1 6.486} C_DIS
LIN {X -0.031,Y -172.850,Z 1583.997,A 0.000,B 0.000,C 90.000,E1 359.542} C_DIS
LIN {X 0.025,Y -174.134,Z 1583.940,A 0.000,B 0.000,C 90.000,E1 349.218} C_DIS
LIN {X -0.017,Y -176.756,Z 1583.912,A 0.000,B 0.000,C 90.000,E1 344.102} C_DIS
LIN {X 0.065,Y -180.103,Z 1583.888,A 0.000,B 0.000,C 90.000,E1 339.826} C_DIS
LIN {X 0.063,Y -184.615,Z 1583.865,A 0.000,B 0.000,C 90.000,E1 335.613} C_DIS
LIN {X 0.039,Y -189.064,Z 1583.846,A 0.000,B 0.000,C 90.000,E1 332.281} C_DIS
LIN {X -0.030,Y -194.175,Z 1583.828,A 0.000,B 0.000,C 90.000,E1 328.997} C_DIS
LIN {X -0.001,Y -200.001,Z 1583.810,A 0.000,B 0.000,C 90.000,E1 325.722} C_DIS
LIN {X 0.074,Y -206.661,Z 1583.792,A 0.000,B 0.000,C 90.000,E1 322.477} C_DIS
LIN {X 0.078,Y -214.186,Z 1583.774,A 0.000,B 0.000,C 90.000,E1 319.299} C_DIS
LIN {X -0.059,Y -222.510,Z 1583.757,A 0.000,B 0.000,C 90.000,E1 316.215} C_DIS
LIN {X 0.001,Y -231.732,Z 1583.740,A 0.000,B 0.000,C 90.000,E1 313.137} C_DIS
LIN {X -0.008,Y -242.121,Z 1583.723,A 0.000,B 0.000,C 90.000,E1 310.135} C_DIS
LIN {X -0.056,Y -248.037,Z 1583.715,A 0.000,B 0.000,C 90.000,E1 308.669} C_DIS
LIN {X -0.029,Y -254.712,Z 1583.707,A 0.000,B 0.000,C 90.000,E1 307.202} C_DIS
LIN {X 0.031,Y -264.068,Z 1583.697,A 0.000,B 0.000,C 90.000,E1 305.391} C_DIS
LIN {X 0.024,Y -274.369,Z 1583.687,A 0.000,B 0.000,C 90.000,E1 303.627} C_DIS
LIN {X 0.075,Y -287.924,Z 1583.675,A 0.000,B 0.000,C 90.000,E1 301.544} C_DIS
LIN {X 0.014,Y -305.154,Z 1583.662,A 0.000,B 0.000,C 90.000,E1 299.205} C_DIS
LIN {X -0.105,Y -317.604,Z 1583.653,A 0.000,B 0.000,C 90.000,E1 297.590} C_DIS
LIN {X -0.072,Y -332.588,Z 1583.643,A 0.000,B 0.000,C 90.000,E1 295.668} C_DIS
LIN {X 0.109,Y -344.742,Z 1583.634,A 0.000,B 0.000,C 90.000,E1 294.079} C_DIS
LIN {X 0.029,Y -364.802,Z 1583.620,A 0.000,B 0.000,C 90.000,E1 291.663} C_DIS
LIN {X 0.099,Y -377.358,Z 1583.612,A 0.000,B 0.000,C 90.000,E1 290.174} C_DIS
LIN {X -0.038,Y -384.556,Z 1583.607,A 0.000,B 0.000,C 90.000,E1 289.322} C_DIS
LIN {X -0.120,Y -391.320,Z 1583.603,A 0.000,B 0.000,C 90.000,E1 288.471} C_DIS
LIN {X 0.120,Y -397.517,Z 1583.598,A 0.000,B 0.000,C 90.000,E1 287.583} C_DIS
LIN {X 0.158,Y -403.083,Z 1583.593,A 0.000,B 0.000,C 90.000,E1 286.732} C_DIS
LIN {X 0.134,Y -407.731,Z 1583.588,A 0.000,B 0.000,C 90.000,E1 285.898} C_DIS
LIN {X 0.147,Y -411.520,Z 1583.584,A 0.000,B 0.000,C 90.000,E1 285.064} C_DIS
LIN {X -0.026,Y -413.577,Z 1583.581,A 0.000,B 0.000,C 90.000,E1 284.537} C_DIS
LIN {X -0.185,Y -415.220,Z 1583.578,A 0.000,B 0.000,C 90.000,E1 284.008} C_DIS
LIN {X 0.165,Y -416.479,Z 1583.575,A 0.000,B 0.000,C 90.000,E1 283.411} C_DIS
LIN {X 0.021,Y -417.334,Z 1583.572,A 0.000,B 0.000,C 90.000,E1 282.883} C_DIS
LIN {X -0.113,Y -417.674,Z 1583.569,A 0.000,B 0.000,C 90.000,E1 282.355} C_DIS
LIN {X 0.164,Y -417.552,Z 1583.566,A 0.000,B 0.000,C 90.000,E1 281.771} C_DIS
LIN {X 0.035,Y -416.910,Z 1583.563,A 0.000,B 0.000,C 90.000,E1 281.243} C_DIS
LIN {X -0.095,Y -415.692,Z 1583.559,A 0.000,B 0.000,C 90.000,E1 280.715} C_DIS
LIN {X 0.103,Y -413.918,Z 1583.556,A 0.000,B 0.000,C 90.000,E1 280.141} C_DIS
LIN {X -0.039,Y -411.426,Z 1583.553,A 0.000,B 0.000,C 90.000,E1 279.613} C_DIS
LIN {X 0.204,Y -408.327,Z 1583.550,A 0.000,B 0.000,C 90.000,E1 279.029} C_DIS
LIN {X -0.037,Y -404.455,Z 1583.547,A 0.000,B 0.000,C 90.000,E1 278.511} C_DIS
LIN {X 0.105,Y -399.900,Z 1583.544,A 0.000,B 0.000,C 90.000,E1 277.936} C_DIS
LIN {X -0.118,Y -394.557,Z 1583.541,A 0.000,B 0.000,C 90.000,E1 277.409} C_DIS
LIN {X 0.132,Y -388.673,Z 1583.538,A 0.000,B 0.000,C 90.000,E1 276.834} C_DIS
LIN {X -0.043,Y -382.670,Z 1583.535,A 0.000,B 0.000,C 90.000,E1 276.372} C_DIS
LIN {X 0.043,Y -376.435,Z 1583.533,A 0.000,B 0.000,C 90.000,E1 275.910} C_DIS
LIN {X 0.010,Y -370.147,Z 1583.531,A 0.000,B 0.000,C 90.000,E1 275.511} C_DIS
LIN {X -0.154,Y -360.561,Z 1583.528,A 0.000,B 0.000,C 90.000,E1 274.992} C_DIS
LIN {X 0.039,Y -350.819,Z 1583.525,A 0.000,B 0.000,C 90.000,E1 274.473} C_DIS
LIN {X -0.153,Y -341.190,Z 1583.522,A 0.000,B 0.000,C 90.000,E1 274.069} C_DIS
LIN {X -0.095,Y -331.515,Z 1583.520,A 0.000,B 0.000,C 90.000,E1 273.669} C_DIS
LIN {X 0.079,Y -318.503,Z 1583.518,A 0.000,B 0.000,C 90.000,E1 273.154} C_DIS
LIN {X -0.090,Y -308.244,Z 1583.516,A 0.000,B 0.000,C 90.000,E1 272.865} C_DIS
LIN {X 0.121,Y -301.201,Z 1583.515,A 0.000,B 0.000,C 90.000,E1 272.636} C_DIS
LIN {X -0.133,Y -293.722,Z 1583.514,A 0.000,B 0.000,C 90.000,E1 272.522} C_DIS
LIN {X 0.017,Y -280.901,Z 1583.513,A 0.000,B 0.000,C 90.000,E1 272.293} C_DIS
LIN {X 0.068,Y -262.562,Z 1583.512,A 0.000,B 0.000,C 90.000,E1 272.064} C_DIS
LIN {X 0.035,Y -245.957,Z 1583.511,A 0.000,B 0.000,C 90.000,E1 271.949} C_DIS
LIN {X -0.054,Y -236.032,Z 1583.511,A 0.000,B 0.000,C 90.000,E1 271.949} C_DIS
LIN {X -0.075,Y -181.274,Z 1583.511,A 0.000,B 0.000,C 90.000,E1 271.949} C_DIS
LIN {X -0.064,Y -181.580,Z 1583.501,A 0.000,B 0.000,C 90.000,E1 270.229} C_DIS
LIN {X -0.074,Y -180.890,Z 1583.473,A 0.000,B 0.000,C 90.000,E1 265.179} C_DIS
LIN {X -0.012,Y -179.014,Z 1583.445,A 0.000,B 0.000,C 90.000,E1 260.095} C_DIS
LIN {X 0.083,Y -178.638,Z 1583.440,A 0.000,B 0.000,C 90.000,E1 259.218} C_DIS
LIN {X -0.020,Y -175.689,Z 1583.412,A 0.000,B 0.000,C 90.000,E1 254.157} C_DIS
LIN {X -0.009,Y -172.405,Z 1583.388,A 0.000,B 0.000,C 90.000,E1 249.880} C_DIS
LIN {X 0.008,Y -171.219,Z 1583.379,A 0.000,B 0.000,C 90.000,E1 248.156} C_DIS
LIN {X -0.016,Y -167.502,Z 1583.355,A 0.000,B 0.000,C 90.000,E1 243.845} C_DIS
LIN {X -0.083,Y -166.897,Z 1583.350,A 0.000,B 0.000,C 90.000,E1 242.999} C_DIS
LIN {X -0.030,Y -162.204,Z 1583.321,A 0.000,B 0.000,C 90.000,E1 237.740} C_DIS
LIN {X 0.023,Y -160.779,Z 1583.311,A 0.000,B 0.000,C 90.000,E1 235.960} C_DIS
LIN {X -0.005,Y -157.572,Z 1583.291,A 0.000,B 0.000,C 90.000,E1 232.431} C_DIS
LIN {X 0.029,Y -155.602,Z 1583.276,A 0.000,B 0.000,C 90.000,E1 229.747} C_DIS
LIN {X 0.079,Y -151.883,Z 1583.251,A 0.000,B 0.000,C 90.000,E1 225.243} C_DIS
LIN {X 0.093,Y -150.109,Z 1583.236,A 0.000,B 0.000,C 90.000,E1 222.528} C_DIS
LIN {X 0.010,Y -146.905,Z 1583.211,A 0.000,B 0.000,C 90.000,E1 218.016} C_DIS
LIN {X -0.090,Y -145.492,Z 1583.196,A 0.000,B 0.000,C 90.000,E1 215.311} C_DIS
LIN {X 0.030,Y -142.899,Z 1583.170,A 0.000,B 0.000,C 90.000,E1 210.669} C_DIS
LIN {X -0.040,Y -141.519,Z 1583.150,A 0.000,B 0.000,C 90.000,E1 207.001} C_DIS
LIN {X 0.004,Y -139.395,Z 1583.114,A 0.000,B 0.000,C 90.000,E1 200.482} C_DIS
LIN {X 0.054,Y -139.105,Z 1583.103,A 0.000,B 0.000,C 90.000,E1 198.598} C_DIS
LIN {X 0.046,Y -138.354,Z 1583.057,A 0.000,B 0.000,C 90.000,E1 190.197} C_DIS
LIN {X 0.039,Y -139.511,Z 1583.005,A 0.000,B 0.000,C 90.000,E1 180.859} C_DIS
LIN {X -0.020,Y -141.157,Z 1582.974,A 0.000,B 0.000,C 90.000,E1 175.298} C_DIS
LIN {X -0.049,Y -142.536,Z 1582.958,A 0.000,B 0.000,C 90.000,E1 172.527} C_DIS
LIN {X 0.019,Y -144.806,Z 1582.933,A 0.000,B 0.000,C 90.000,E1 167.881} C_DIS
LIN {X 0.007,Y -147.426,Z 1582.912,A 0.000,B 0.000,C 90.000,E1 164.212} C_DIS
LIN {X 0.035,Y -150.003,Z 1582.892,A 0.000,B 0.000,C 90.000,E1 160.550} C_DIS
LIN {X 0.042,Y -153.334,Z 1582.872,A 0.000,B 0.000,C 90.000,E1 156.922} C_DIS
LIN {X 0.024,Y -155.870,Z 1582.857,A 0.000,B 0.000,C 90.000,E1 154.229} C_DIS
LIN {X -0.009,Y -159.723,Z 1582.837,A 0.000,B 0.000,C 90.000,E1 150.667} C_DIS
LIN {X 0.057,Y -161.962,Z 1582.827,A 0.000,B 0.000,C 90.000,E1 148.869} C_DIS
LIN {X -0.058,Y -166.153,Z 1582.808,A 0.000,B 0.000,C 90.000,E1 145.388} C_DIS
LIN {X -0.064,Y -171.165,Z 1582.788,A 0.000,B 0.000,C 90.000,E1 141.904} C_DIS
LIN {X -0.029,Y -176.046,Z 1582.769,A 0.000,B 0.000,C 90.000,E1 138.447} C_DIS
LIN {X -0.034,Y -180.300,Z 1582.755,A 0.000,B 0.000,C 90.000,E1 135.891} C_DIS
LIN {X -0.062,Y -185.713,Z 1582.736,A 0.000,B 0.000,C 90.000,E1 132.528} C_DIS
LIN {X -0.010,Y -190.319,Z 1582.722,A 0.000,B 0.000,C 90.000,E1 130.011} C_DIS
LIN {X 0.038,Y -197.645,Z 1582.699,A 0.000,B 0.000,C 90.000,E1 125.884} C_DIS
LIN {X -0.033,Y -200.902,Z 1582.690,A 0.000,B 0.000,C 90.000,E1 124.278} C_DIS
LIN {X 0.050,Y -204.382,Z 1582.679,A 0.000,B 0.000,C 90.000,E1 122.291} C_DIS
LIN {X 0.042,Y -321.514,Z 1582.679,A 0.000,B 0.000,C 90.000,E1 122.291} C_DIS
LIN {X -0.056,Y -327.781,Z 1582.678,A 0.000,B 0.000,C 90.000,E1 122.084} C_DIS
LIN {X -0.157,Y -330.558,Z 1582.677,A 0.000,B 0.000,C 90.000,E1 121.878} C_DIS
LIN {X -0.020,Y -334.320,Z 1582.674,A 0.000,B 0.000,C 90.000,E1 121.386} C_DIS
LIN {X 0.101,Y -336.077,Z 1582.673,A 0.000,B 0.000,C 90.000,E1 121.052} C_DIS
LIN {X 0.018,Y -343.750,Z 1582.662,A 0.000,B 0.000,C 90.000,E1 119.205} C_DIS
LIN {X -0.156,Y -356.186,Z 1582.647,A 0.000,B 0.000,C 90.000,E1 116.488} C_DIS
LIN {X 0.039,Y -370.107,Z 1582.632,A 0.000,B 0.000,C 90.000,E1 113.770} C_DIS
LIN {X -0.146,Y -383.830,Z 1582.619,A 0.000,B 0.000,C 90.000,E1 111.461} C_DIS
LIN {X 0.085,Y -398.919,Z 1582.606,A 0.000,B 0.000,C 90.000,E1 109.141} C_DIS
LIN {X 0.060,Y -415.478,Z 1582.594,A 0.000,B 0.000,C 90.000,E1 106.913} C_DIS
LIN {X -0.205,Y -433.623,Z 1582.582,A 0.000,B 0.000,C 90.000,E1 104.773} C_DIS
LIN {X 0.041,Y -453.241,Z 1582.570,A 0.000,B 0.000,C 90.000,E1 102.647} C_DIS
LIN {X 0.043,Y -473.527,Z 1582.560,A 0.000,B 0.000,C 90.000,E1 100.715} C_DIS
LIN {X 0.231,Y -494.297,Z 1582.550,A 0.000,B 0.000,C 90.000,E1 98.916} C_DIS
LIN {X -0.141,Y -496.391,Z 1582.548,A 0.000,B 0.000,C 90.000,E1 98.746} C_DIS
LIN {X -0.221,Y -498.194,Z 1582.547,A 0.000,B 0.000,C 90.000,E1 98.511} C_DIS
LIN {X 0.191,Y -499.542,Z 1582.546,A 0.000,B 0.000,C 90.000,E1 98.219} C_DIS
LIN {X -0.032,Y -501.218,Z 1582.543,A 0.000,B 0.000,C 90.000,E1 97.757} C_DIS
LIN {X 0.250,Y -501.794,Z 1582.540,A 0.000,B 0.000,C 90.000,E1 97.239} C_DIS
LIN {X 0.044,Y -501.370,Z 1582.538,A 0.000,B 0.000,C 90.000,E1 96.777} C_DIS
LIN {X -0.158,Y -499.879,Z 1582.535,A 0.000,B 0.000,C 90.000,E1 96.315} C_DIS
LIN {X 0.210,Y -498.654,Z 1582.534,A 0.000,B 0.000,C 90.000,E1 96.030} C_DIS
LIN {X -0.081,Y -482.383,Z 1582.520,A 0.000,B 0.000,C 90.000,E1 93.612} C_DIS
LIN {X -0.128,Y -472.478,Z 1582.512,A 0.000,B 0.000,C 90.000,E1 92.121} C_DIS
LIN {X -0.134,Y -463.926,Z 1582.505,A 0.000,B 0.000,C 90.000,E1 90.859} C_DIS
LIN {X -0.043,Y -453.138,Z 1582.496,A 0.000,B 0.000,C 90.000,E1 89.312} C_DIS
LIN {X 0.120,Y -443.716,Z 1582.489,A 0.000,B 0.000,C 90.000,E1 87.993} C_DIS
LIN {X 0.151,Y -433.829,Z 1582.482,A 0.000,B 0.000,C 90.000,E1 86.674} C_DIS
LIN {X 0.024,Y -417.808,Z 1582.470,A 0.000,B 0.000,C 90.000,E1 84.546} C_DIS
LIN {X -0.117,Y -395.109,Z 1582.451,A 0.000,B 0.000,C 90.000,E1 81.254} C_DIS
LIN {X -0.130,Y -377.567,Z 1582.436,A 0.000,B 0.000,C 90.000,E1 78.409} C_DIS
LIN {X 0.002,Y -361.012,Z 1582.419,A 0.000,B 0.000,C 90.000,E1 75.463} C_DIS
LIN {X -0.054,Y -349.757,Z 1582.408,A 0.000,B 0.000,C 90.000,E1 73.378} C_DIS
LIN {X -0.039,Y -334.173,Z 1582.391,A 0.000,B 0.000,C 90.000,E1 70.315} C_DIS
LIN {X 0.047,Y -322.306,Z 1582.377,A 0.000,B 0.000,C 90.000,E1 67.794} C_DIS
LIN {X 0.091,Y -310.840,Z 1582.362,A 0.000,B 0.000,C 90.000,E1 65.229} C_DIS
LIN {X 0.112,Y -299.850,Z 1582.348,A 0.000,B 0.000,C 90.000,E1 62.615} C_DIS
LIN {X -0.109,Y -291.581,Z 1582.337,A 0.000,B 0.000,C 90.000,E1 60.667} C_DIS
LIN {X 0.055,Y -283.110,Z 1582.326,A 0.000,B 0.000,C 90.000,E1 58.614} C_DIS
LIN {X 0.058,Y -273.094,Z 1582.312,A 0.000,B 0.000,C 90.000,E1 56.215} C_DIS
LIN {X -0.005,Y -263.118,Z 1582.299,A 0.000,B 0.000,C 90.000,E1 53.783} C_DIS
LIN {X 0.041,Y -250.883,Z 1582.281,A 0.000,B 0.000,C 90.000,E1 50.561} C_DIS
LIN {X -0.118,Y -239.510,Z 1582.263,A 0.000,B 0.000,C 90.000,E1 47.310} C_DIS
LIN {X -0.108,Y -229.184,Z 1582.244,A 0.000,B 0.000,C 90.000,E1 43.947} C_DIS
LIN {X 0.053,Y -220.838,Z 1582.227,A 0.000,B 0.000,C 90.000,E1 40.862} C_DIS
LIN {X -0.105,Y -213.183,Z 1582.210,A 0.000,B 0.000,C 90.000,E1 37.810} C_DIS
LIN {X 0.090,Y -206.347,Z 1582.192,A 0.000,B 0.000,C 90.000,E1 34.612} C_DIS
LIN {X -0.066,Y -200.243,Z 1582.175,A 0.000,B 0.000,C 90.000,E1 31.465} C_DIS
LIN {X -0.061,Y -194.978,Z 1582.157,A 0.000,B 0.000,C 90.000,E1 28.231} C_DIS
LIN {X -0.038,Y -189.402,Z 1582.134,A 0.000,B 0.000,C 90.000,E1 24.131} C_DIS
LIN {X -0.052,Y -184.722,Z 1582.111,A 0.000,B 0.000,C 90.000,E1 19.993} C_DIS
LIN {X 0.009,Y -180.883,Z 1582.088,A 0.000,B 0.000,C 90.000,E1 15.788} C_DIS
LIN {X 0.021,Y -177.296,Z 1582.060,A 0.000,B 0.000,C 90.000,E1 10.715} C_DIS
LIN {X -0.035,Y -174.819,Z 1582.031,A 0.000,B 0.000,C 90.000,E1 5.625} C_DIS
LIN {X -0.021,Y -172.917,Z 1581.983,A 0.000,B 0.000,C 90.000,E1 356.963} C_DIS
LIN {X -0.066,Y -174.738,Z 1581.935,A 0.000,B 0.000,C 90.000,E1 348.398} C_DIS
LIN {X -0.045,Y -177.600,Z 1581.907,A 0.000,B 0.000,C 90.000,E1 343.268} C_DIS
LIN {X -0.049,Y -181.145,Z 1581.883,A 0.000,B 0.000,C 90.000,E1 339.028} C_DIS
LIN {X 0.053,Y -185.871,Z 1581.860,A 0.000,B 0.000,C 90.000,E1 334.793} C_DIS
LIN {X -0.110,Y -190.463,Z 1581.842,A 0.000,B 0.000,C 90.000,E1 331.513} C_DIS
LIN {X -0.054,Y -195.727,Z 1581.823,A 0.000,B 0.000,C 90.000,E1 328.201} C_DIS
LIN {X 0.122,Y -201.713,Z 1581.805,A 0.000,B 0.000,C 90.000,E1 324.895} C_DIS
LIN {X 0.073,Y -208.556,Z 1581.787,A 0.000,B 0.000,C 90.000,E1 321.698} C_DIS
LIN {X 0.007,Y -217.295,Z 1581.768,A 0.000,B 0.000,C 90.000,E1 318.162} C_DIS
LIN {X -0.059,Y -225.849,Z 1581.750,A 0.000,B 0.000,C 90.000,E1 315.081} C_DIS
LIN {X 0.102,Y -235.442,Z 1581.734,A 0.000,B 0.000,C 90.000,E1 312.000} C_DIS
LIN {X -0.093,Y -243.432,Z 1581.721,A 0.000,B 0.000,C 90.000,E1 309.806} C_DIS
LIN {X 0.034,Y -249.525,Z 1581.713,A 0.000,B 0.000,C 90.000,E1 308.302} C_DIS
LIN {X -0.071,Y -256.352,Z 1581.705,A 0.000,B 0.000,C 90.000,E1 306.870} C_DIS
LIN {X 0.072,Y -267.885,Z 1581.693,A 0.000,B 0.000,C 90.000,E1 304.692} C_DIS
LIN {X -0.083,Y -280.785,Z 1581.681,A 0.000,B 0.000,C 90.000,E1 302.625} C_DIS
LIN {X 0.087,Y -297.517,Z 1581.668,A 0.000,B 0.000,C 90.000,E1 300.207} C_DIS
LIN {X 0.040,Y -312.457,Z 1581.657,A 0.000,B 0.000,C 90.000,E1 298.231} C_DIS
LIN {X -0.021,Y -327.437,Z 1581.646,A 0.000,B 0.000,C 90.000,E1 296.309} C_DIS
LIN {X 0.082,Y -339.762,Z 1581.637,A 0.000,B 0.000,C 90.000,E1 294.719} C_DIS
LIN {X 0.136,Y -362.115,Z 1581.622,A 0.000,B 0.000,C 90.000,E1 291.972} C_DIS
LIN {X -0.160,Y -374.591,Z 1581.614,A 0.000,B 0.000,C 90.000,E1 290.556} C_DIS
LIN {X -0.205,Y -384.369,Z 1581.608,A 0.000,B 0.000,C 90.000,E1 289.396} C_DIS
LIN {X 0.083,Y -391.188,Z 1581.603,A 0.000,B 0.000,C 90.000,E1 288.489} C_DIS
LIN {X 0.073,Y -397.455,Z 1581.598,A 0.000,B 0.000,C 90.000,E1 287.638} C_DIS
LIN {X -0.075,Y -401.305,Z 1581.595,A 0.000,B 0.000,C 90.000,E1 287.094} C_DIS
LIN {X -0.124,Y -406.295,Z 1581.590,A 0.000,B 0.000,C 90.000,E1 286.260} C_DIS
LIN {X 0.172,Y -409.188,Z 1581.587,A 0.000,B 0.000,C 90.000,E1 285.662} C_DIS
LIN {X 0.204,Y -412.713,Z 1581.583,A 0.000,B 0.000,C 90.000,E1 284.828} C_DIS
LIN {X -0.082,Y -413.741,Z 1581.581,A 0.000,B 0.000,C 90.000,E1 284.592} C_DIS
LIN {X 0.162,Y -415.460,Z 1581.578,A 0.000,B 0.000,C 90.000,E1 284.008} C_DIS
LIN {X 0.011,Y -416.790,Z 1581.575,A 0.000,B 0.000,C 90.000,E1 283.480} C_DIS
LIN {X -0.034,Y -417.672,Z 1581.572,A 0.000,B 0.000,C 90.000,E1 282.939} C_DIS
LIN {X -0.169,Y -418.087,Z 1581.569,A 0.000,B 0.000,C 90.000,E1 282.411} C_DIS
LIN {X 0.110,Y -418.021,Z 1581.566,A 0.000,B 0.000,C 90.000,E1 281.827} C_DIS
LIN {X -0.017,Y -417.445,Z 1581.563,A 0.000,B 0.000,C 90.000,E1 281.299} C_DIS
LIN {X -0.223,Y -416.293,Z 1581.560,A 0.000,B 0.000,C 90.000,E1 280.782} C_DIS
LIN {X 0.055,Y -414.586,Z 1581.557,A 0.000,B 0.000,C 90.000,E1 280.197} C_DIS
LIN {X -0.083,Y -412.191,Z 1581.554,A 0.000,B 0.000,C 90.000,E1 279.670} C_DIS
LIN {X 0.100,Y -409.193,Z 1581.551,A 0.000,B 0.000,C 90.000,E1 279.095} C_DIS
LIN {X -0.073,Y -405.411,Z 1581.547,A 0.000,B 0.000,C 90.000,E1 278.568} C_DIS
LIN {X 0.074,Y -400.867,Z 1581.544,A 0.000,B 0.000,C 90.000,E1 277.992} C_DIS
LIN {X -0.144,Y -395.624,Z 1581.541,A 0.000,B 0.000,C 90.000,E1 277.466} C_DIS
LIN {X 0.151,Y -389.897,Z 1581.538,A 0.000,B 0.000,C 90.000,E1 276.891} C_DIS
LIN {X -0.024,Y -383.965,Z 1581.536,A 0.000,B 0.000,C 90.000,E1 276.429} C_DIS
LIN {X 0.058,Y -377.758,Z 1581.533,A 0.000,B 0.000,C 90.000,E1 275.967} C_DIS
LIN {X -0.068,Y -368.382,Z 1581.530,A 0.000,B 0.000,C 90.000,E1 275.391} C_DIS
LIN {X -0.184,Y -361.968,Z 1581.528,A 0.000,B 0.000,C 90.000,E1 275.049} C_DIS
LIN {X 0.024,Y -352.314,Z 1581.525,A 0.000,B 0.000,C 90.000,E1 274.531} C_DIS
LIN {X 0.121,Y -342.653,Z 1581.523,A 0.000,B 0.000,C 90.000,E1 274.073} C_DIS
LIN {X 0.074,Y -329.578,Z 1581.520,A 0.000,B 0.000,C 90.000,E1 273.555} C_DIS
LIN {X -0.062,Y -319.686,Z 1581.518,A 0.000,B 0.000,C 90.000,E1 273.212} C_DIS
LIN {X 0.092,Y -309.559,Z 1581.516,A 0.000,B 0.000,C 90.000,E1 272.865} C_DIS
LIN {X 0.135,Y -298.919,Z 1581.515,A 0.000,B 0.000,C 90.000,E1 272.579} C_DIS
LIN {X -0.085,Y -291.203,Z 1581.514,A 0.000,B 0.000,C 90.000,E1 272.465} C_DIS
LIN {X -0.139,Y -273.649,Z 1581.512,A 0.000,B 0.000,C 90.000,E1 272.236} C_DIS
LIN {X -0.035,Y -260.122,Z 1581.511,A 0.000,B 0.000,C 90.000,E1 272.064} C_DIS
LIN {X 0.056,Y -246.101,Z 1581.511,A 0.000,B 0.000,C 90.000,E1 271.949} C_DIS
LIN {X 0.009,Y -240.044,Z 1581.511,A 0.000,B 0.000,C 90.000,E1 271.949} C_DIS
LIN {X -0.035,Y -233.238,Z 1581.511,A 0.000,B 0.000,C 90.000,E1 271.949} C_DIS
LIN {X -0.062,Y -181.274,Z 1581.511,A 0.000,B 0.000,C 90.000,E1 271.949} C_DIS
LIN {X 0.010,Y -181.576,Z 1581.502,A 0.000,B 0.000,C 90.000,E1 270.401} C_DIS
LIN {X -0.029,Y -180.910,Z 1581.476,A 0.000,B 0.000,C 90.000,E1 265.698} C_DIS
LIN {X 0.029,Y -180.820,Z 1581.471,A 0.000,B 0.000,C 90.000,E1 264.837} C_DIS
LIN {X -0.071,Y -178.924,Z 1581.443,A 0.000,B 0.000,C 90.000,E1 259.803} C_DIS
LIN {X -0.033,Y -175.970,Z 1581.415,A 0.000,B 0.000,C 90.000,E1 254.700} C_DIS
LIN {X -0.038,Y -175.453,Z 1581.410,A 0.000,B 0.000,C 90.000,E1 253.850} C_DIS
LIN {X -0.030,Y -172.206,Z 1581.386,A 0.000,B 0.000,C 90.000,E1 249.571} C_DIS
LIN {X -0.052,Y -171.680,Z 1581.382,A 0.000,B 0.000,C 90.000,E1 248.720} C_DIS
LIN {X -0.061,Y -167.906,Z 1581.358,A 0.000,B 0.000,C 90.000,E1 244.409} C_DIS
LIN {X -0.042,Y -166.647,Z 1581.348,A 0.000,B 0.000,C 90.000,E1 242.666} C_DIS
LIN {X 0.012,Y -162.631,Z 1581.324,A 0.000,B 0.000,C 90.000,E1 238.280} C_DIS
LIN {X 0.071,Y -161.319,Z 1581.314,A 0.000,B 0.000,C 90.000,E1 236.501} C_DIS
LIN {X -0.020,Y -157.314,Z 1581.289,A 0.000,B 0.000,C 90.000,E1 232.110} C_DIS
LIN {X -0.087,Y -155.294,Z 1581.275,A 0.000,B 0.000,C 90.000,E1 229.461} C_DIS
LIN {X 0.060,Y -151.655,Z 1581.250,A 0.000,B 0.000,C 90.000,E1 224.919} C_DIS
LIN {X -0.003,Y -150.522,Z 1581.240,A 0.000,B 0.000,C 90.000,E1 223.137} C_DIS
LIN {X 0.020,Y -147.247,Z 1581.214,A 0.000,B 0.000,C 90.000,E1 218.588} C_DIS
LIN {X -0.015,Y -145.272,Z 1581.194,A 0.000,B 0.000,C 90.000,E1 214.945} C_DIS
LIN {X 0.019,Y -142.379,Z 1581.163,A 0.000,B 0.000,C 90.000,E1 209.411} C_DIS
LIN {X 0.069,Y -141.354,Z 1581.148,A 0.000,B 0.000,C 90.000,E1 206.616} C_DIS
LIN {X 0.051,Y -139.340,Z 1581.112,A 0.000,B 0.000,C 90.000,E1 200.120} C_DIS
LIN {X -0.030,Y -139.008,Z 1581.102,A 0.000,B 0.000,C 90.000,E1 198.290} C_DIS
LIN {X 0.057,Y -138.340,Z 1581.055,A 0.000,B 0.000,C 90.000,E1 189.849} C_DIS
LIN {X -0.059,Y -139.403,Z 1581.008,A 0.000,B 0.000,C 90.000,E1 181.489} C_DIS
LIN {X -0.006,Y -141.308,Z 1580.972,A 0.000,B 0.000,C 90.000,E1 174.951} C_DIS
LIN {X -0.048,Y -142.668,Z 1580.956,A 0.000,B 0.000,C 90.000,E1 172.186} C_DIS
LIN {X 0.073,Y -145.017,Z 1580.931,A 0.000,B 0.000,C 90.000,E1 167.521} C_DIS
LIN {X 0.031,Y -147.644,Z 1580.910,A 0.000,B 0.000,C 90.000,E1 163.866} C_DIS
LIN {X -0.033,Y -150.277,Z 1580.890,A 0.000,B 0.000,C 90.000,E1 160.242} C_DIS
LIN {X -0.021,Y -153.681,Z 1580.870,A 0.000,B 0.000,C 90.000,E1 156.613} C_DIS
LIN {X 0.035,Y -157.095,Z 1580.850,A 0.000,B 0.000,C 90.000,E1 152.999} C_DIS
LIN {X -0.027,Y -161.232,Z 1580.830,A 0.000,B 0.000,C 90.000,E1 149.459} C_DIS
LIN {X 0.059,Y -163.321,Z 1580.820,A 0.000,B 0.000,C 90.000,E1 147.661} C_DIS
LIN {X -0.071,Y -167.773,Z 1580.801,A 0.000,B 0.000,C 90.000,E1 144.196} C_DIS
LIN {X 0.082,Y -171.588,Z 1580.786,A 0.000,B 0.000,C 90.000,E1 141.537} C_DIS
LIN {X 0.012,Y -176.538,Z 1580.767,A 0.000,B 0.000,C 90.000,E1 138.119} C_DIS
LIN {X 0.005,Y -180.837,Z 1580.753,A 0.000,B 0.000,C 90.000,E1 135.567} C_DIS
LIN {X -0.010,Y -186.247,Z 1580.734,A 0.000,B 0.000,C 90.000,E1 132.204} C_DIS
LIN {X -0.073,Y -190.883,Z 1580.721,A 0.000,B 0.000,C 90.000,E1 129.725} C_DIS
LIN {X -0.040,Y -196.647,Z 1580.702,A 0.000,B 0.000,C 90.000,E1 126.423} C_DIS
LIN {X 0.036,Y -199.888,Z 1580.693,A 0.000,B 0.000,C 90.000,E1 124.771} C_DIS
LIN {X 0.022,Y -204.306,Z 1580.680,A 0.000,B 0.000,C 90.000,E1 122.339} C_DIS
LIN {X 0.000,Y -320.696,Z 1580.680,A 0.000,B 0.000,C 90.000,E1 122.339} C_DIS
LIN {X 0.030,Y -323.632,Z 1580.679,A 0.000,B 0.000,C 90.000,E1 122.291} C_DIS
LIN {X -0.124,Y -327.638,Z 1580.678,A 0.000,B 0.000,C 90.000,E1 122.133} C_DIS
LIN {X -0.002,Y -330.000,Z 1580.677,A 0.000,B 0.000,C 90.000,E1 121.926} C_DIS
LIN {X 0.071,Y -333.243,Z 1580.675,A 0.000,B 0.000,C 90.000,E1 121.544} C_DIS
LIN {X -0.043,Y -335.159,Z 1580.674,A 0.000,B 0.000,C 90.000,E1 121.258} C_DIS
LIN {X 0.129,Y -336.652,Z 1580.672,A 0.000,B 0.000,C 90.000,E1 120.924} C_DIS
LIN {X 0.097,Y -349.612,Z 1580.655,A 0.000,B 0.000,C 90.000,E1 117.847} C_DIS
LIN {X -0.060,Y -362.756,Z 1580.640,A 0.000,B 0.000,C 90.000,E1 115.155} C_DIS
LIN {X 0.176,Y -377.450,Z 1580.625,A 0.000,B 0.000,C 90.000,E1 112.461} C_DIS
LIN {X 0.031,Y -391.910,Z 1580.612,A 0.000,B 0.000,C 90.000,E1 110.174} C_DIS
LIN {X -0.170,Y -407.793,Z 1580.600,A 0.000,B 0.000,C 90.000,E1 107.946} C_DIS
LIN {X 0.020,Y -425.207,Z 1580.587,A 0.000,B 0.000,C 90.000,E1 105.717} C_DIS
LIN {X -0.111,Y -444.261,Z 1580.575,A 0.000,B 0.000,C 90.000,E1 103.592} C_DIS
LIN {X -0.168,Y -464.293,Z 1580.564,A 0.000,B 0.000,C 90.000,E1 101.591} C_DIS
LIN {X 0.052,Y -487.460,Z 1580.553,A 0.000,B 0.000,C 90.000,E1 99.500} C_DIS
LIN {X -0.009,Y -495.151,Z 1580.549,A 0.000,B 0.000,C 90.000,E1 98.859} C_DIS
LIN {X 0.096,Y -497.083,Z 1580.548,A 0.000,B 0.000,C 90.000,E1 98.624} C_DIS
LIN {X 0.126,Y -498.558,Z 1580.547,A 0.000,B 0.000,C 90.000,E1 98.398} C_DIS
LIN {X 0.049,Y -499.779,Z 1580.545,A 0.000,B 0.000,C 90.000,E1 98.163} C_DIS
LIN {X -0.100,Y -500.664,Z 1580.544,A 0.000,B 0.000,C 90.000,E1 97.936} C_DIS
LIN {X 0.250,Y -501.587,Z 1580.541,A 0.000,B 0.000,C 90.000,E1 97.409} C_DIS
LIN {X 0.040,Y -501.497,Z 1580.539,A 0.000,B 0.000,C 90.000,E1 96.947} C_DIS
LIN {X -0.165,Y -500.383,Z 1580.536,A 0.000,B 0.000,C 90.000,E1 96.486} C_DIS
LIN {X 0.202,Y -499.390,Z 1580.535,A 0.000,B 0.000,C 90.000,E1 96.201} C_DIS
LIN {X 0.126,Y -498.040,Z 1580.533,A 0.000,B 0.000,C 90.000,E1 95.967} C_DIS
LIN {X -0.229,Y -481.741,Z 1580.520,A 0.000,B 0.000,C 90.000,E1 93.555} C_DIS
LIN {X 0.190,Y -471.831,Z 1580.511,A 0.000,B 0.000,C 90.000,E1 92.007} C_DIS
LIN {X 0.164,Y -463.266,Z 1580.504,A 0.000,B 0.000,C 90.000,E1 90.745} C_DIS
LIN {X -0.216,Y -452.458,Z 1580.496,A 0.000,B 0.000,C 90.000,E1 89.255} C_DIS
LIN {X -0.054,Y -442.997,Z 1580.489,A 0.000,B 0.000,C 90.000,E1 87.936} C_DIS
LIN {X 0.121,Y -431.102,Z 1580.480,A 0.000,B 0.000,C 90.000,E1 86.331} C_DIS
LIN {X 0.055,Y -413.218,Z 1580.466,A 0.000,B 0.000,C 90.000,E1 83.913} C_DIS
LIN {X 0.135,Y -390.874,Z 1580.448,A 0.000,B 0.000,C 90.000,E1 80.566} C_DIS
LIN {X 0.122,Y -373.599,Z 1580.432,A 0.000,B 0.000,C 90.000,E1 77.701} C_DIS
LIN {X 0.174,Y -358.834,Z 1580.417,A 0.000,B 0.000,C 90.000,E1 75.046} C_DIS
LIN {X -0.007,Y -346.014,Z 1580.404,A 0.000,B 0.000,C 90.000,E1 72.670} C_DIS
LIN {X 0.105,Y -330.651,Z 1580.387,A 0.000,B 0.000,C 90.000,E1 69.571} C_DIS
LIN {X 0.046,Y -317.465,Z 1580.371,A 0.000,B 0.000,C 90.000,E1 66.741} C_DIS
LIN {X 0.031,Y -303.378,Z 1580.353,A 0.000,B 0.000,C 90.000,E1 63.512} C_DIS
LIN {X 0.137,Y -295.118,Z 1580.342,A 0.000,B 0.000,C 90.000,E1 61.513} C_DIS
LIN {X -0.028,Y -286.742,Z 1580.331,A 0.000,B 0.000,C 90.000,E1 59.537} C_DIS
LIN {X -0.090,Y -276.772,Z 1580.318,A 0.000,B 0.000,C 90.000,E1 57.168} C_DIS
LIN {X 0.080,Y -268.248,Z 1580.306,A 0.000,B 0.000,C 90.000,E1 55.055} C_DIS
LIN {X -0.056,Y -255.743,Z 1580.288,A 0.000,B 0.000,C 90.000,E1 51.904} C_DIS
LIN {X -0.054,Y -244.055,Z 1580.270,A 0.000,B 0.000,C 90.000,E1 48.647} C_DIS
LIN {X -0.095,Y -233.288,Z 1580.252,A 0.000,B 0.000,C 90.000,E1 45.324} C_DIS
LIN {X -0.075,Y -223.569,Z 1580.233,A 0.000,B 0.000,C 90.000,E1 41.919} C_DIS
LIN {X -0.026,Y -215.722,Z 1580.216,A 0.000,B 0.000,C 90.000,E1 38.830} C_DIS
LIN {X 0.063,Y -208.591,Z 1580.198,A 0.000,B 0.000,C 90.000,E1 35.678} C_DIS
LIN {X -0.093,Y -202.287,Z 1580.181,A 0.000,B 0.000,C 90.000,E1 32.546} C_DIS
LIN {X 0.061,Y -196.748,Z 1580.163,A 0.000,B 0.000,C 90.000,E1 29.283} C_DIS
LIN {X 0.052,Y -190.922,Z 1580.140,A 0.000,B 0.000,C 90.000,E1 25.207} C_DIS
LIN {X -0.017,Y -186.053,Z 1580.117,A 0.000,B 0.000,C 90.000,E1 21.099} C_DIS
LIN {X 0.023,Y -182.015,Z 1580.094,A 0.000,B 0.000,C 90.000,E1 16.913} C_DIS
LIN {X -0.059,Y -178.208,Z 1580.066,A 0.000,B 0.000,C 90.000,E1 11.883} C_DIS
LIN {X 0.009,Y -175.154,Z 1580.033,A 0.000,B 0.000,C 90.000,E1 5.910} C_DIS
LIN {X -0.019,Y -173.176,Z 1579.988,A 0.000,B 0.000,C 90.000,E1 357.822} C_DIS
LIN {X 0.061,Y -174.640,Z 1579.940,A 0.000,B 0.000,C 90.000,E1 349.218} C_DIS
LIN {X 0.038,Y -177.284,Z 1579.912,A 0.000,B 0.000,C 90.000,E1 344.102} C_DIS
LIN {X -0.031,Y -180.602,Z 1579.888,A 0.000,B 0.000,C 90.000,E1 339.880} C_DIS
LIN {X -0.016,Y -185.085,Z 1579.865,A 0.000,B 0.000,C 90.000,E1 335.665} C_DIS
LIN {X -0.113,Y -189.452,Z 1579.846,A 0.000,B 0.000,C 90.000,E1 332.359} C_DIS
LIN {X 0.087,Y -194.512,Z 1579.828,A 0.000,B 0.000,C 90.000,E1 328.997} C_DIS
LIN {X 0.014,Y -200.288,Z 1579.810,A 0.000,B 0.000,C 90.000,E1 325.754} C_DIS
LIN {X -0.077,Y -206.865,Z 1579.792,A 0.000,B 0.000,C 90.000,E1 322.557} C_DIS
LIN {X -0.074,Y -214.366,Z 1579.774,A 0.000,B 0.000,C 90.000,E1 319.380} C_DIS
LIN {X -0.139,Y -223.679,Z 1579.755,A 0.000,B 0.000,C 90.000,E1 315.891} C_DIS
LIN {X 0.119,Y -232.929,Z 1579.738,A 0.000,B 0.000,C 90.000,E1 312.771} C_DIS
LIN {X 0.010,Y -241.948,Z 1579.723,A 0.000,B 0.000,C 90.000,E1 310.172} C_DIS
LIN {X -0.035,Y -247.819,Z 1579.715,A 0.000,B 0.000,C 90.000,E1 308.705} C_DIS
LIN {X -0.005,Y -254.424,Z 1579.707,A 0.000,B 0.000,C 90.000,E1 307.237} C_DIS
LIN {X -0.058,Y -267.713,Z 1579.693,A 0.000,B 0.000,C 90.000,E1 304.739} C_DIS
LIN {X 0.008,Y -280.607,Z 1579.681,A 0.000,B 0.000,C 90.000,E1 302.625} C_DIS
LIN {X -0.079,Y -299.804,Z 1579.666,A 0.000,B 0.000,C 90.000,E1 299.922} C_DIS
LIN {X 0.134,Y -312.253,Z 1579.657,A 0.000,B 0.000,C 90.000,E1 298.231} C_DIS
LIN {X 0.074,Y -327.272,Z 1579.646,A 0.000,B 0.000,C 90.000,E1 296.309} C_DIS
LIN {X -0.132,Y -339.634,Z 1579.637,A 0.000,B 0.000,C 90.000,E1 294.771} C_DIS
LIN {X -0.091,Y -364.694,Z 1579.621,A 0.000,B 0.000,C 90.000,E1 291.716} C_DIS
LIN {X -0.141,Y -377.336,Z 1579.612,A 0.000,B 0.000,C 90.000,E1 290.248} C_DIS
LIN {X -0.038,Y -386.866,Z 1579.606,A 0.000,B 0.000,C 90.000,E1 289.087} C_DIS
LIN {X -0.091,Y -393.520,Z 1579.601,A 0.000,B 0.000,C 90.000,E1 288.236} C_DIS
LIN {X -0.214,Y -399.629,Z 1579.597,A 0.000,B 0.000,C 90.000,E1 287.402} C_DIS
LIN {X 0.036,Y -403.296,Z 1579.593,A 0.000,B 0.000,C 90.000,E1 286.804} C_DIS
LIN {X -0.075,Y -406.562,Z 1579.590,A 0.000,B 0.000,C 90.000,E1 286.260} C_DIS
LIN {X -0.069,Y -410.719,Z 1579.586,A 0.000,B 0.000,C 90.000,E1 285.426} C_DIS
LIN {X -0.030,Y -414.028,Z 1579.581,A 0.000,B 0.000,C 90.000,E1 284.592} C_DIS
LIN {X -0.187,Y -415.789,Z 1579.578,A 0.000,B 0.000,C 90.000,E1 284.064} C_DIS
LIN {X 0.068,Y -417.136,Z 1579.575,A 0.000,B 0.000,C 90.000,E1 283.480} C_DIS
LIN {X 0.025,Y -418.037,Z 1579.572,A 0.000,B 0.000,C 90.000,E1 282.939} C_DIS
LIN {X -0.108,Y -418.517,Z 1579.569,A 0.000,B 0.000,C 90.000,E1 282.411} C_DIS
LIN {X 0.173,Y -418.475,Z 1579.566,A 0.000,B 0.000,C 90.000,E1 281.827} C_DIS
LIN {X 0.049,Y -417.903,Z 1579.563,A 0.000,B 0.000,C 90.000,E1 281.299} C_DIS
LIN {X -0.156,Y -416.796,Z 1579.560,A 0.000,B 0.000,C 90.000,E1 280.782} C_DIS
LIN {X 0.126,Y -415.145,Z 1579.557,A 0.000,B 0.000,C 90.000,E1 280.197} C_DIS
LIN {X -0.010,Y -412.782,Z 1579.554,A 0.000,B 0.000,C 90.000,E1 279.670} C_DIS
LIN {X 0.175,Y -409.778,Z 1579.551,A 0.000,B 0.000,C 90.000,E1 279.095} C_DIS
LIN {X 0.005,Y -406.078,Z 1579.548,A 0.000,B 0.000,C 90.000,E1 278.568} C_DIS
LIN {X 0.156,Y -401.587,Z 1579.545,A 0.000,B 0.000,C 90.000,E1 277.992} C_DIS
LIN {X -0.060,Y -396.333,Z 1579.541,A 0.000,B 0.000,C 90.000,E1 277.466} C_DIS
LIN {X 0.187,Y -390.521,Z 1579.538,A 0.000,B 0.000,C 90.000,E1 276.891} C_DIS
LIN {X 0.012,Y -384.539,Z 1579.536,A 0.000,B 0.000,C 90.000,E1 276.429} C_DIS
LIN {X 0.108,Y -378.404,Z 1579.533,A 0.000,B 0.000,C 90.000,E1 275.967} C_DIS
LIN {X -0.016,Y -368.972,Z 1579.530,A 0.000,B 0.000,C 90.000,E1 275.391} C_DIS
LIN {X -0.118,Y -362.573,Z 1579.528,A 0.000,B 0.000,C 90.000,E1 275.049} C_DIS
LIN {X 0.097,Y -352.910,Z 1579.525,A 0.000,B 0.000,C 90.000,E1 274.531} C_DIS
LIN {X -0.129,Y -343.302,Z 1579.523,A 0.000,B 0.000,C 90.000,E1 274.131} C_DIS
LIN {X 0.149,Y -330.187,Z 1579.520,A 0.000,B 0.000,C 90.000,E1 273.555} C_DIS
LIN {X 0.024,Y -320.334,Z 1579.518,A 0.000,B 0.000,C 90.000,E1 273.212} C_DIS
LIN {X -0.120,Y -310.219,Z 1579.516,A 0.000,B 0.000,C 90.000,E1 272.922} C_DIS
LIN {X -0.102,Y -299.561,Z 1579.515,A 0.000,B 0.000,C 90.000,E1 272.636} C_DIS
LIN {X -0.044,Y -291.875,Z 1579.514,A 0.000,B 0.000,C 90.000,E1 272.465} C_DIS
LIN {X -0.134,Y -278.525,Z 1579.513,A 0.000,B 0.000,C 90.000,E1 272.293} C_DIS
LIN {X -0.009,Y -260.525,Z 1579.511,A 0.000,B 0.000,C 90.000,E1 272.064} C_DIS
LIN {X 0.076,Y -246.298,Z 1579.511,A 0.000,B 0.000,C 90.000,E1 271.949} C_DIS
LIN {X 0.028,Y -239.234,Z 1579.511,A 0.000,B 0.000,C 90.000,E1 271.949} C_DIS
LIN {X -0.017,Y -231.499,Z 1579.511,A 0.000,B 0.000,C 90.000,E1 271.949} C_DIS
LIN {X -0.048,Y -181.272,Z 1579.511,A 0.000,B 0.000,C 90.000,E1 271.949} C_DIS
LIN {X 0.024,Y -181.576,Z 1579.502,A 0.000,B 0.000,C 90.000,E1 270.401} C_DIS
LIN {X -0.015,Y -180.910,Z 1579.476,A 0.000,B 0.000,C 90.000,E1 265.698} C_DIS
LIN {X 0.042,Y -180.821,Z 1579.471,A 0.000,B 0.000,C 90.000,E1 264.837} C_DIS
LIN {X -0.058,Y -178.925,Z 1579.443,A 0.000,B 0.000,C 90.000,E1 259.803} C_DIS
LIN {X -0.018,Y -175.972,Z 1579.415,A 0.000,B 0.000,C 90.000,E1 254.700} C_DIS
LIN {X -0.025,Y -175.456,Z 1579.410,A 0.000,B 0.000,C 90.000,E1 253.850} C_DIS
LIN {X -0.016,Y -172.208,Z 1579.386,A 0.000,B 0.000,C 90.000,E1 249.571} C_DIS
LIN {X -0.039,Y -171.684,Z 1579.382,A 0.000,B 0.000,C 90.000,E1 248.720} C_DIS
LIN {X -0.048,Y -167.910,Z 1579.358,A 0.000,B 0.000,C 90.000,E1 244.409} C_DIS
LIN {X -0.030,Y -166.651,Z 1579.348,A 0.000,B 0.000,C 90.000,E1 242.666} C_DIS
LIN {X 0.025,Y -162.635,Z 1579.324,A 0.000,B 0.000,C 90.000,E1 238.280} C_DIS
LIN {X -0.050,Y -161.322,Z 1579.314,A 0.000,B 0.000,C 90.000,E1 236.548} C_DIS
LIN {X -0.007,Y -157.318,Z 1579.289,A 0.000,B 0.000,C 90.000,E1 232.110} C_DIS
LIN {X -0.074,Y -155.298,Z 1579.275,A 0.000,B 0.000,C 90.000,E1 229.461} C_DIS
LIN {X 0.072,Y -151.658,Z 1579.250,A 0.000,B 0.000,C 90.000,E1 224.919} C_DIS
LIN {X 0.009,Y -150.525,Z 1579.240,A 0.000,B 0.000,C 90.000,E1 223.137} C_DIS
LIN {X 0.032,Y -147.250,Z 1579.214,A 0.000,B 0.000,C 90.000,E1 218.588} C_DIS
LIN {X -0.003,Y -145.275,Z 1579.194,A 0.000,B 0.000,C 90.000,E1 214.945} C_DIS
LIN {X 0.032,Y -142.380,Z 1579.163,A 0.000,B 0.000,C 90.000,E1 209.411} C_DIS
LIN {X -0.046,Y -141.357,Z 1579.148,A 0.000,B 0.000,C 90.000,E1 206.668} C_DIS
LIN {X 0.063,Y -139.341,Z 1579.112,A 0.000,B 0.000,C 90.000,E1 200.120} C_DIS
LIN {X -0.019,Y -139.010,Z 1579.102,A 0.000,B 0.000,C 90.000,E1 198.290} C_DIS
LIN {X -0.067,Y -138.341,Z 1579.055,A 0.000,B 0.000,C 90.000,E1 189.905} C_DIS
LIN {X -0.047,Y -139.401,Z 1579.008,A 0.000,B 0.000,C 90.000,E1 181.489} C_DIS
LIN {X 0.006,Y -141.306,Z 1578.972,A 0.000,B 0.000,C 90.000,E1 174.951} C_DIS
LIN {X -0.036,Y -142.666,Z 1578.957,A 0.000,B 0.000,C 90.000,E1 172.186} C_DIS
LIN {X 0.055,Y -145.014,Z 1578.931,A 0.000,B 0.000,C 90.000,E1 167.533} C_DIS
LIN {X 0.043,Y -147.641,Z 1578.910,A 0.000,B 0.000,C 90.000,E1 163.866} C_DIS
LIN {X -0.021,Y -150.273,Z 1578.890,A 0.000,B 0.000,C 90.000,E1 160.242} C_DIS
LIN {X -0.008,Y -153.675,Z 1578.870,A 0.000,B 0.000,C 90.000,E1 156.613} C_DIS
LIN {X 0.048,Y -157.090,Z 1578.850,A 0.000,B 0.000,C 90.000,E1 152.999} C_DIS
LIN {X -0.014,Y -161.227,Z 1578.830,A 0.000,B 0.000,C 90.000,E1 149.459} C_DIS
LIN {X 0.072,Y -163.316,Z 1578.820,A 0.000,B 0.000,C 90.000,E1 147.661} C_DIS
LIN {X -0.057,Y -167.766,Z 1578.801,A 0.000,B 0.000,C 90.000,E1 144.196} C_DIS
LIN {X 0.095,Y -171.581,Z 1578.786,A 0.000,B 0.000,C 90.000,E1 141.537} C_DIS
LIN {X -0.106,Y -176.531,Z 1578.767,A 0.000,B 0.000,C 90.000,E1 138.162} C_DIS
LIN {X 0.019,Y -180.830,Z 1578.753,A 0.000,B 0.000,C 90.000,E1 135.567} C_DIS
LIN {X 0.004,Y -186.239,Z 1578.734,A 0.000,B 0.000,C 90.000,E1 132.204} C_DIS
LIN {X -0.058,Y -190.876,Z 1578.721,A 0.000,B 0.000,C 90.000,E1 129.725} C_DIS
LIN {X -0.026,Y -196.640,Z 1578.702,A 0.000,B 0.000,C 90.000,E1 126.423} C_DIS
LIN {X -0.113,Y -199.880,Z 1578.693,A 0.000,B 0.000,C 90.000,E1 124.818} C_DIS
LIN {X -0.113,Y -204.230,Z 1578.680,A 0.000,B 0.000,C 90.000,E1 122.418} C_DIS
LIN {X -0.051,Y -320.452,Z 1578.680,A 0.000,B 0.000,C 90.000,E1 122.388} C_DIS
LIN {X 0.130,Y -322.236,Z 1578.680,A 0.000,B 0.000,C 90.000,E1 122.339} C_DIS
LIN {X -0.070,Y -325.076,Z 1578.679,A 0.000,B 0.000,C 90.000,E1 122.291} C_DIS
LIN {X 0.041,Y -328.298,Z 1578.678,A 0.000,B 0.000,C 90.000,E1 122.084} C_DIS
LIN {X -0.064,Y -331.957,Z 1578.676,A 0.000,B 0.000,C 90.000,E1 121.750} C_DIS
LIN {X -0.055,Y -335.464,Z 1578.673,A 0.000,B 0.000,C 90.000,E1 121.209} C_DIS
LIN {X -0.094,Y -338.117,Z 1578.670,A 0.000,B 0.000,C 90.000,E1 120.590} C_DIS
LIN {X 0.210,Y -349.857,Z 1578.654,A 0.000,B 0.000,C 90.000,E1 117.769} C_DIS
LIN {X 0.052,Y -363.036,Z 1578.639,A 0.000,B 0.000,C 90.000,E1 115.079} C_DIS
LIN {X -0.197,Y -377.761,Z 1578.625,A 0.000,B 0.000,C 90.000,E1 112.461} C_DIS
LIN {X 0.020,Y -392.254,Z 1578.612,A 0.000,B 0.000,C 90.000,E1 110.120} C_DIS
LIN {X -0.042,Y -408.172,Z 1578.599,A 0.000,B 0.000,C 90.000,E1 107.873} C_DIS
LIN {X 0.037,Y -425.624,Z 1578.587,A 0.000,B 0.000,C 90.000,E1 105.662} C_DIS
LIN {X -0.067,Y -444.706,Z 1578.575,A 0.000,B 0.000,C 90.000,E1 103.536} C_DIS
LIN {X -0.088,Y -464.753,Z 1578.564,A 0.000,B 0.000,C 90.000,E1 101.535} C_DIS
LIN {X 0.155,Y -487.960,Z 1578.553,A 0.000,B 0.000,C 90.000,E1 99.443} C_DIS
LIN {X 0.001,Y -493.198,Z 1578.550,A 0.000,B 0.000,C 90.000,E1 99.029} C_DIS
LIN {X 0.127,Y -495.494,Z 1578.549,A 0.000,B 0.000,C 90.000,E1 98.803} C_DIS
LIN {X -0.161,Y -497.231,Z 1578.548,A 0.000,B 0.000,C 90.000,E1 98.624} C_DIS
LIN {X 0.176,Y -498.759,Z 1578.547,A 0.000,B 0.000,C 90.000,E1 98.341} C_DIS
LIN {X 0.094,Y -499.896,Z 1578.545,A 0.000,B 0.000,C 90.000,E1 98.106} C_DIS
LIN {X -0.125,Y -501.234,Z 1578.542,A 0.000,B 0.000,C 90.000,E1 97.644} C_DIS
LIN {X 0.160,Y -501.523,Z 1578.540,A 0.000,B 0.000,C 90.000,E1 97.125} C_DIS
LIN {X -0.044,Y -500.808,Z 1578.537,A 0.000,B 0.000,C 90.000,E1 96.663} C_DIS
LIN {X -0.247,Y -498.973,Z 1578.534,A 0.000,B 0.000,C 90.000,E1 96.201} C_DIS
LIN {X 0.043,Y -495.841,Z 1578.532,A 0.000,B 0.000,C 90.000,E1 95.682} C_DIS
LIN {X -0.194,Y -481.240,Z 1578.519,A 0.000,B 0.000,C 90.000,E1 93.498} C_DIS
LIN {X 0.214,Y -471.325,Z 1578.511,A 0.000,B 0.000,C 90.000,E1 91.949} C_DIS
LIN {X 0.186,Y -462.763,Z 1578.504,A 0.000,B 0.000,C 90.000,E1 90.688} C_DIS
LIN {X 0.024,Y -453.784,Z 1578.497,A 0.000,B 0.000,C 90.000,E1 89.427} C_DIS
LIN {X 0.199,Y -444.413,Z 1578.490,A 0.000,B 0.000,C 90.000,E1 88.108} C_DIS
LIN {X -0.200,Y -434.575,Z 1578.482,A 0.000,B 0.000,C 90.000,E1 86.846} C_DIS
LIN {X 0.084,Y -418.597,Z 1578.470,A 0.000,B 0.000,C 90.000,E1 84.666} C_DIS
LIN {X -0.051,Y -395.823,Z 1578.452,A 0.000,B 0.000,C 90.000,E1 81.376} C_DIS
LIN {X 0.043,Y -376.548,Z 1578.435,A 0.000,B 0.000,C 90.000,E1 78.229} C_DIS
LIN {X 0.081,Y -361.642,Z 1578.420,A 0.000,B 0.000,C 90.000,E1 75.589} C_DIS
LIN {X 0.066,Y -348.789,Z 1578.407,A 0.000,B 0.000,C 90.000,E1 73.196} C_DIS
LIN {X 0.172,Y -334.759,Z 1578.391,A 0.000,B 0.000,C 90.000,E1 70.423} C_DIS
LIN {X 0.056,Y -319.958,Z 1578.374,A 0.000,B 0.000,C 90.000,E1 67.305} C_DIS
LIN {X -0.162,Y -309.895,Z 1578.361,A 0.000,B 0.000,C 90.000,E1 65.101} C_DIS
LIN {X -0.154,Y -298.818,Z 1578.347,A 0.000,B 0.000,C 90.000,E1 62.487} C_DIS
LIN {X 0.004,Y -289.064,Z 1578.334,A 0.000,B 0.000,C 90.000,E1 60.127} C_DIS
LIN {X -0.120,Y -280.532,Z 1578.323,A 0.000,B 0.000,C 90.000,E1 58.122} C_DIS
LIN {X 0.060,Y -270.688,Z 1578.309,A 0.000,B 0.000,C 90.000,E1 55.674} C_DIS
LIN {X 0.151,Y -259.461,Z 1578.294,A 0.000,B 0.000,C 90.000,E1 52.844} C_DIS
LIN {X 0.091,Y -247.535,Z 1578.276,A 0.000,B 0.000,C 90.000,E1 49.622} C_DIS
LIN {X -0.020,Y -236.491,Z 1578.257,A 0.000,B 0.000,C 90.000,E1 46.338} C_DIS
LIN {X 0.076,Y -226.483,Z 1578.239,A 0.000,B 0.000,C 90.000,E1 42.933} C_DIS
LIN {X 0.028,Y -218.417,Z 1578.222,A 0.000,B 0.000,C 90.000,E1 39.886} C_DIS
LIN {X -0.023,Y -211.054,Z 1578.204,A 0.000,B 0.000,C 90.000,E1 36.790} C_DIS
LIN {X -0.007,Y -204.474,Z 1578.187,A 0.000,B 0.000,C 90.000,E1 33.627} C_DIS
LIN {X 0.026,Y -198.669,Z 1578.169,A 0.000,B 0.000,C 90.000,E1 30.413} C_DIS
LIN {X -0.010,Y -193.715,Z 1578.151,A 0.000,B 0.000,C 90.000,E1 27.180} C_DIS
LIN {X -0.004,Y -189.404,Z 1578.133,A 0.000,B 0.000,C 90.000,E1 23.898} C_DIS
LIN {X -0.011,Y -184.839,Z 1578.110,A 0.000,B 0.000,C 90.000,E1 19.758} C_DIS
LIN {X 0.058,Y -181.066,Z 1578.087,A 0.000,B 0.000,C 90.000,E1 15.552} C_DIS
LIN {X 0.043,Y -177.605,Z 1578.058,A 0.000,B 0.000,C 90.000,E1 10.489} C_DIS
LIN {X 0.024,Y -175.162,Z 1578.030,A 0.000,B 0.000,C 90.000,E1 5.391} C_DIS
LIN {X -0.003,Y -173.420,Z 1577.978,A 0.000,B 0.000,C 90.000,E1 356.102} C_DIS
LIN {X -0.062,Y -175.248,Z 1577.936,A 0.000,B 0.000,C 90.000,E1 348.409} C_DIS
LIN {X 0.013,Y -178.131,Z 1577.907,A 0.000,B 0.000,C 90.000,E1 343.268} C_DIS
LIN {X 0.027,Y -181.661,Z 1577.884,A 0.000,B 0.000,C 90.000,E1 339.028} C_DIS
LIN {X -0.021,Y -186.353,Z 1577.860,A 0.000,B 0.000,C 90.000,E1 334.845} C_DIS
LIN {X -0.003,Y -190.843,Z 1577.842,A 0.000,B 0.000,C 90.000,E1 331.513} C_DIS
LIN {X 0.065,Y -196.048,Z 1577.823,A 0.000,B 0.000,C 90.000,E1 328.201} C_DIS
LIN {X -0.028,Y -201.975,Z 1577.805,A 0.000,B 0.000,C 90.000,E1 324.975} C_DIS
LIN {X 0.051,Y -208.758,Z 1577.788,A 0.000,B 0.000,C 90.000,E1 321.743} C_DIS
LIN {X -0.147,Y -217.453,Z 1577.768,A 0.000,B 0.000,C 90.000,E1 318.243} C_DIS
LIN {X 0.028,Y -227.028,Z 1577.748,A 0.000,B 0.000,C 90.000,E1 314.717} C_DIS
LIN {X 0.056,Y -236.646,Z 1577.732,A 0.000,B 0.000,C 90.000,E1 311.676} C_DIS
LIN {X 0.082,Y -243.255,Z 1577.721,A 0.000,B 0.000,C 90.000,E1 309.806} C_DIS
LIN {X 0.057,Y -249.270,Z 1577.713,A 0.000,B 0.000,C 90.000,E1 308.338} C_DIS
LIN {X 0.084,Y -254.285,Z 1577.707,A 0.000,B 0.000,C 90.000,E1 307.237} C_DIS
LIN {X 0.032,Y -267.538,Z 1577.693,A 0.000,B 0.000,C 90.000,E1 304.739} C_DIS
LIN {X 0.099,Y -280.437,Z 1577.681,A 0.000,B 0.000,C 90.000,E1 302.625} C_DIS
LIN {X 0.015,Y -299.608,Z 1577.666,A 0.000,B 0.000,C 90.000,E1 299.922} C_DIS
LIN {X -0.047,Y -312.059,Z 1577.657,A 0.000,B 0.000,C 90.000,E1 298.281} C_DIS
LIN {X -0.124,Y -327.105,Z 1577.646,A 0.000,B 0.000,C 90.000,E1 296.360} C_DIS
LIN {X -0.036,Y -339.505,Z 1577.638,A 0.000,B 0.000,C 90.000,E1 294.771} C_DIS
LIN {X -0.074,Y -362.081,Z 1577.622,A 0.000,B 0.000,C 90.000,E1 292.025} C_DIS
LIN {X -0.175,Y -374.888,Z 1577.614,A 0.000,B 0.000,C 90.000,E1 290.556} C_DIS
LIN {X -0.167,Y -384.733,Z 1577.608,A 0.000,B 0.000,C 90.000,E1 289.396} C_DIS
LIN {X 0.124,Y -391.616,Z 1577.603,A 0.000,B 0.000,C 90.000,E1 288.489} C_DIS
LIN {X 0.118,Y -397.906,Z 1577.598,A 0.000,B 0.000,C 90.000,E1 287.638} C_DIS
LIN {X 0.042,Y -403.565,Z 1577.593,A 0.000,B 0.000,C 90.000,E1 286.804} C_DIS
LIN {X -0.070,Y -406.846,Z 1577.590,A 0.000,B 0.000,C 90.000,E1 286.260} C_DIS
LIN {X -0.164,Y -409.737,Z 1577.587,A 0.000,B 0.000,C 90.000,E1 285.717} C_DIS
LIN {X 0.045,Y -412.243,Z 1577.584,A 0.000,B 0.000,C 90.000,E1 285.134} C_DIS
LIN {X -0.017,Y -414.355,Z 1577.581,A 0.000,B 0.000,C 90.000,E1 284.592} C_DIS
LIN {X -0.174,Y -416.132,Z 1577.578,A 0.000,B 0.000,C 90.000,E1 284.064} C_DIS
LIN {X 0.083,Y -417.509,Z 1577.575,A 0.000,B 0.000,C 90.000,E1 283.480} C_DIS
LIN {X 0.042,Y -418.427,Z 1577.572,A 0.000,B 0.000,C 90.000,E1 282.939} C_DIS
LIN {X -0.089,Y -418.920,Z 1577.569,A 0.000,B 0.000,C 90.000,E1 282.411} C_DIS
LIN {X 0.196,Y -418.939,Z 1577.566,A 0.000,B 0.000,C 90.000,E1 281.827} C_DIS
LIN {X 0.072,Y -418.372,Z 1577.563,A 0.000,B 0.000,C 90.000,E1 281.299} C_DIS
LIN {X -0.129,Y -417.309,Z 1577.560,A 0.000,B 0.000,C 90.000,E1 280.782} C_DIS
LIN {X 0.156,Y -415.669,Z 1577.557,A 0.000,B 0.000,C 90.000,E1 280.197} C_DIS
LIN {X 0.022,Y -413.325,Z 1577.554,A 0.000,B 0.000,C 90.000,E1 279.670} C_DIS
LIN {X -0.194,Y -410.332,Z 1577.551,A 0.000,B 0.000,C 90.000,E1 279.151} C_DIS
LIN {X 0.044,Y -406.706,Z 1577.548,A 0.000,B 0.000,C 90.000,E1 278.568} C_DIS
LIN {X -0.201,Y -402.211,Z 1577.545,A 0.000,B 0.000,C 90.000,E1 278.049} C_DIS
LIN {X -0.016,Y -396.958,Z 1577.542,A 0.000,B 0.000,C 90.000,E1 277.466} C_DIS
LIN {X -0.126,Y -391.256,Z 1577.538,A 0.000,B 0.000,C 90.000,E1 276.947} C_DIS
LIN {X 0.049,Y -385.153,Z 1577.536,A 0.000,B 0.000,C 90.000,E1 276.429} C_DIS
LIN {X 0.158,Y -379.033,Z 1577.533,A 0.000,B 0.000,C 90.000,E1 275.967} C_DIS
LIN {X 0.034,Y -369.597,Z 1577.530,A 0.000,B 0.000,C 90.000,E1 275.391} C_DIS
LIN {X -0.020,Y -359.969,Z 1577.527,A 0.000,B 0.000,C 90.000,E1 274.878} C_DIS
LIN {X 0.001,Y -350.429,Z 1577.525,A 0.000,B 0.000,C 90.000,E1 274.416} C_DIS
LIN {X -0.129,Y -340.834,Z 1577.522,A 0.000,B 0.000,C 90.000,E1 274.012} C_DIS
LIN {X -0.106,Y -324.860,Z 1577.519,A 0.000,B 0.000,C 90.000,E1 273.383} C_DIS
LIN {X -0.062,Y -314.638,Z 1577.517,A 0.000,B 0.000,C 90.000,E1 273.037} C_DIS
LIN {X -0.074,Y -304.513,Z 1577.515,A 0.000,B 0.000,C 90.000,E1 272.751} C_DIS
LIN {X -0.087,Y -297.170,Z 1577.514,A 0.000,B 0.000,C 90.000,E1 272.579} C_DIS
LIN {X 0.035,Y -289.473,Z 1577.513,A 0.000,B 0.000,C 90.000,E1 272.407} C_DIS
LIN {X 0.036,Y -271.729,Z 1577.512,A 0.000,B 0.000,C 90.000,E1 272.178} C_DIS
LIN {X -0.129,Y -256.970,Z 1577.511,A 0.000,B 0.000,C 90.000,E1 272.064} C_DIS
LIN {X 0.119,Y -247.568,Z 1577.511,A 0.000,B 0.000,C 90.000,E1 271.949} C_DIS
LIN {X 0.018,Y -234.169,Z 1577.511,A 0.000,B 0.000,C 90.000,E1 271.949} C_DIS
LIN {X -0.004,Y -181.270,Z 1577.511,A 0.000,B 0.000,C 90.000,E1 271.949} C_DIS
LIN {X 0.084,Y -181.573,Z 1577.502,A 0.000,B 0.000,C 90.000,E1 270.401} C_DIS
LIN {X 0.045,Y -180.910,Z 1577.476,A 0.000,B 0.000,C 90.000,E1 265.698} C_DIS
LIN {X -0.077,Y -180.828,Z 1577.471,A 0.000,B 0.000,C 90.000,E1 264.894} C_DIS
LIN {X 0.003,Y -178.932,Z 1577.443,A 0.000,B 0.000,C 90.000,E1 259.803} C_DIS
LIN {X 0.040,Y -175.980,Z 1577.415,A 0.000,B 0.000,C 90.000,E1 254.700} C_DIS
LIN {X -0.015,Y -175.472,Z 1577.410,A 0.000,B 0.000,C 90.000,E1 253.866} C_DIS
LIN {X 0.043,Y -172.220,Z 1577.387,A 0.000,B 0.000,C 90.000,E1 249.571} C_DIS
LIN {X 0.020,Y -171.697,Z 1577.382,A 0.000,B 0.000,C 90.000,E1 248.720} C_DIS
END
